REGION Network 73: Reset CMS
   // Reset Axis when the unit is in the resetting state.
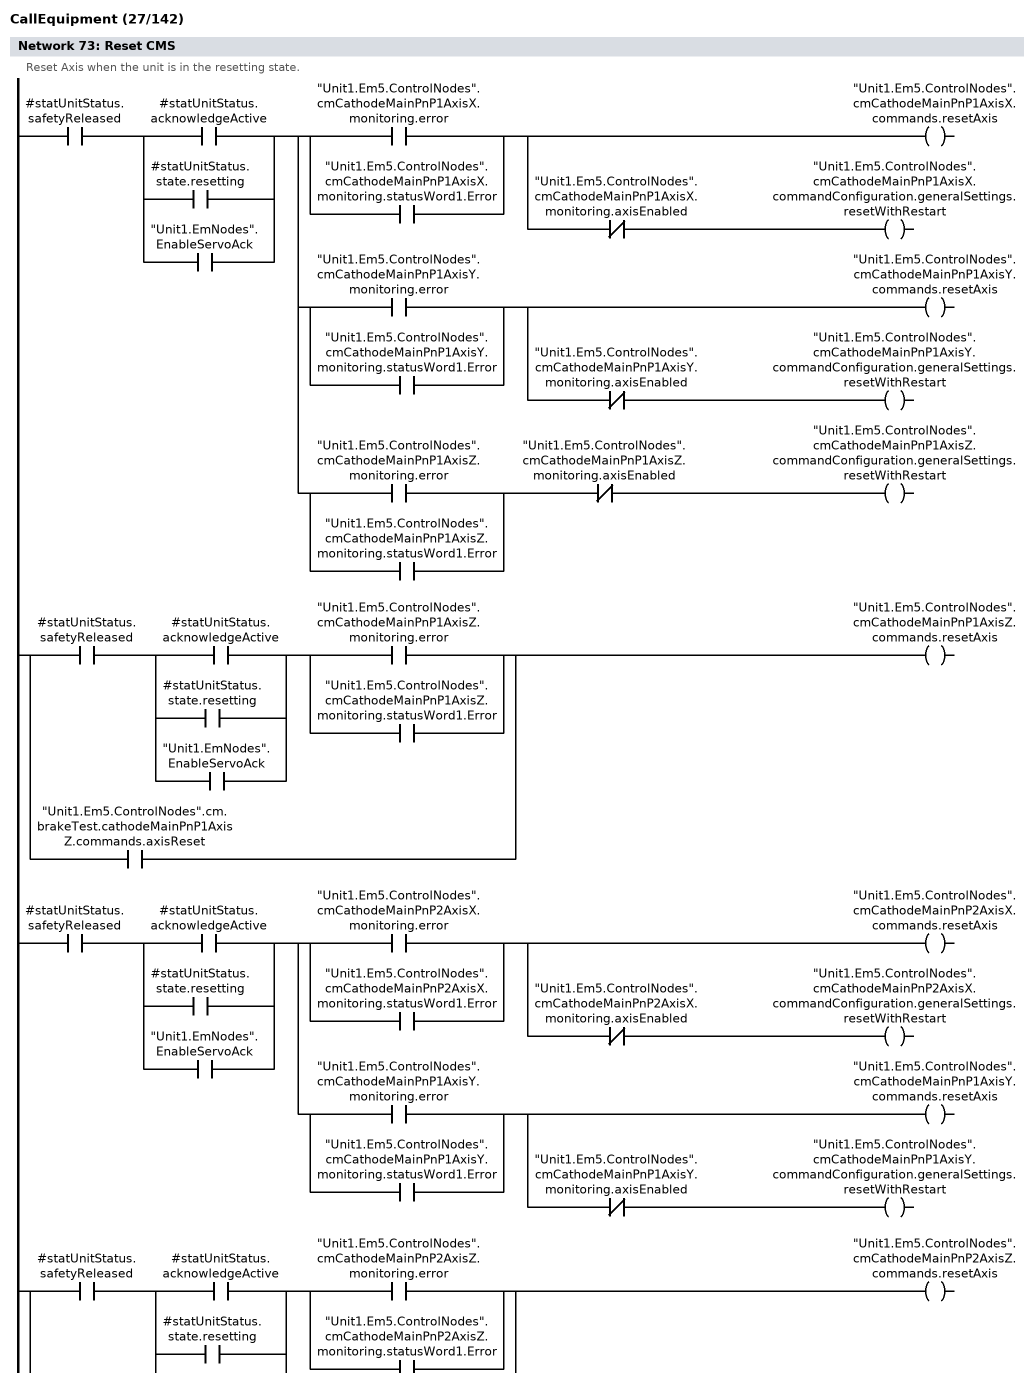
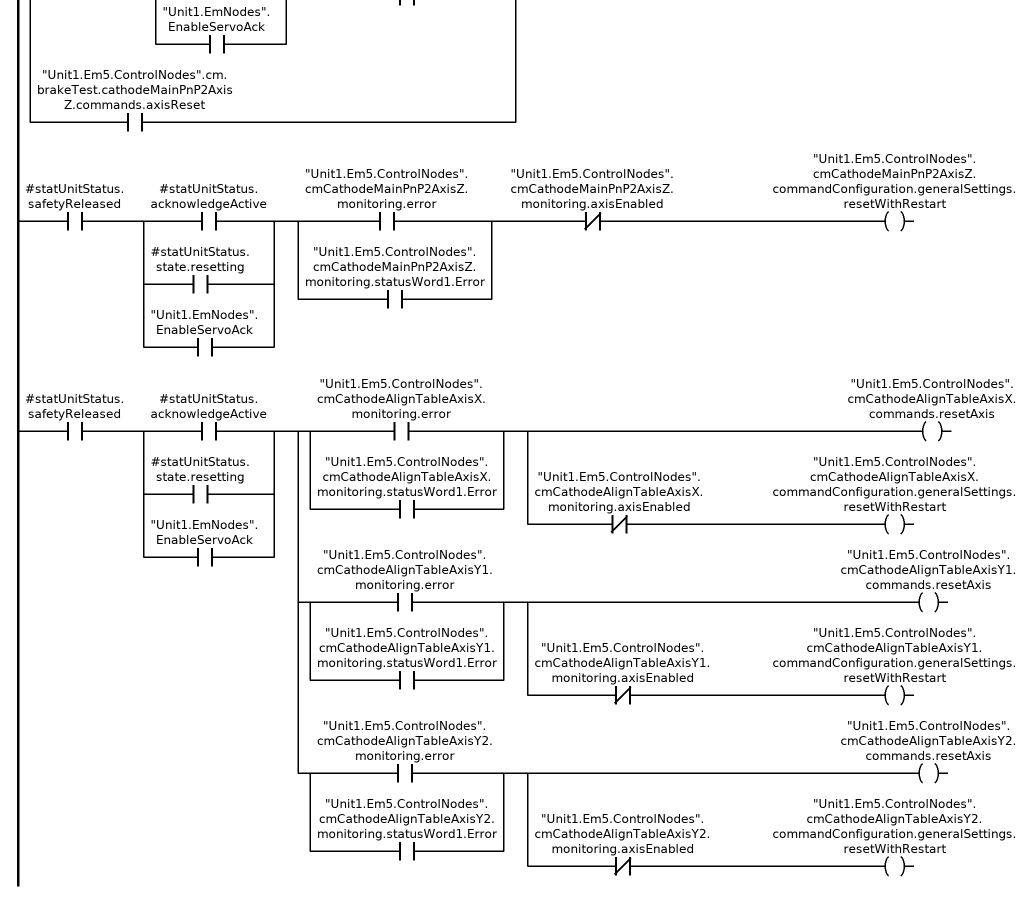
   RUNG wire#powerrail
      Contact( #statUnitStatus.safetyReleased )
      wire#w1
      Contact( #statUnitStatus.acknowledgeActive )
      wire#w2
      Contact( "Unit1.Em5.ControlNodes".cmCathodeMainPnP1AxisX.monitoring.error )
      wire#w3
      Coil( "Unit1.Em5.ControlNodes".cmCathodeMainPnP1AxisX.commands.resetAxis )
   END_RUNG
   RUNG wire#w1
      Contact( #statUnitStatus.state.resetting )
   END_RUNG wire#w2
   RUNG wire#w1
      Contact( "Unit1.EmNodes".EnableServoAck )
   END_RUNG wire#w2
   RUNG wire#w2
      Contact( "Unit1.Em5.ControlNodes".cmCathodeMainPnP1AxisX.monitoring.statusWord1.Error )
   END_RUNG wire#w3
   RUNG wire#w3
      I_Contact( "Unit1.Em5.ControlNodes".cmCathodeMainPnP1AxisX.monitoring.axisEnabled )
      Coil( "Unit1.Em5.ControlNodes".cmCathodeMainPnP1AxisX.commandConfiguration.generalSettings.resetWithRestart )
   END_RUNG
   RUNG wire#w2
      Contact( "Unit1.Em5.ControlNodes".cmCathodeMainPnP1AxisY.monitoring.error )
      wire#w4
      Coil( "Unit1.Em5.ControlNodes".cmCathodeMainPnP1AxisY.commands.resetAxis )
   END_RUNG
   RUNG wire#w2
      Contact( "Unit1.Em5.ControlNodes".cmCathodeMainPnP1AxisY.monitoring.statusWord1.Error )
   END_RUNG wire#w4
   RUNG wire#w4
      I_Contact( "Unit1.Em5.ControlNodes".cmCathodeMainPnP1AxisY.monitoring.axisEnabled )
      Coil( "Unit1.Em5.ControlNodes".cmCathodeMainPnP1AxisY.commandConfiguration.generalSettings.resetWithRestart )
   END_RUNG
   RUNG wire#w2
      Contact( "Unit1.Em5.ControlNodes".cmCathodeMainPnP1AxisZ.monitoring.error )
      wire#w5
      I_Contact( "Unit1.Em5.ControlNodes".cmCathodeMainPnP1AxisZ.monitoring.axisEnabled )
      Coil( "Unit1.Em5.ControlNodes".cmCathodeMainPnP1AxisZ.commandConfiguration.generalSettings.resetWithRestart )
   END_RUNG
   RUNG wire#w2
      Contact( "Unit1.Em5.ControlNodes".cmCathodeMainPnP1AxisZ.monitoring.statusWord1.Error )
   END_RUNG wire#w5
   RUNG wire#powerrail
      Contact( #statUnitStatus.safetyReleased )
      wire#w6
      Contact( #statUnitStatus.acknowledgeActive )
      wire#w7
      Contact( "Unit1.Em5.ControlNodes".cmCathodeMainPnP1AxisZ.monitoring.error )
      wire#w8
      Coil( "Unit1.Em5.ControlNodes".cmCathodeMainPnP1AxisZ.commands.resetAxis )
   END_RUNG
   RUNG wire#w6
      Contact( #statUnitStatus.state.resetting )
   END_RUNG wire#w7
   RUNG wire#w6
      Contact( "Unit1.EmNodes".EnableServoAck )
   END_RUNG wire#w7
   RUNG wire#w7
      Contact( "Unit1.Em5.ControlNodes".cmCathodeMainPnP1AxisZ.monitoring.statusWord1.Error )
   END_RUNG wire#w8
   RUNG wire#powerrail
      Contact( "Unit1.Em5.ControlNodes".cm.brakeTest.cathodeMainPnP1AxisZ.commands.axisReset )
   END_RUNG wire#w8
   RUNG wire#powerrail
      Contact( #statUnitStatus.safetyReleased )
      wire#w9
      Contact( #statUnitStatus.acknowledgeActive )
      wire#w10
      Contact( "Unit1.Em5.ControlNodes".cmCathodeMainPnP2AxisX.monitoring.error )
      wire#w11
      Coil( "Unit1.Em5.ControlNodes".cmCathodeMainPnP2AxisX.commands.resetAxis )
   END_RUNG
   RUNG wire#w9
      Contact( #statUnitStatus.state.resetting )
   END_RUNG wire#w10
   RUNG wire#w9
      Contact( "Unit1.EmNodes".EnableServoAck )
   END_RUNG wire#w10
   RUNG wire#w10
      Contact( "Unit1.Em5.ControlNodes".cmCathodeMainPnP2AxisX.monitoring.statusWord1.Error )
   END_RUNG wire#w11
   RUNG wire#w11
      I_Contact( "Unit1.Em5.ControlNodes".cmCathodeMainPnP2AxisX.monitoring.axisEnabled )
      Coil( "Unit1.Em5.ControlNodes".cmCathodeMainPnP2AxisX.commandConfiguration.generalSettings.resetWithRestart )
   END_RUNG
   RUNG wire#w10
      Contact( "Unit1.Em5.ControlNodes".cmCathodeMainPnP1AxisY.monitoring.error )
      wire#w12
      Coil( "Unit1.Em5.ControlNodes".cmCathodeMainPnP1AxisY.commands.resetAxis )
   END_RUNG
   RUNG wire#w10
      Contact( "Unit1.Em5.ControlNodes".cmCathodeMainPnP1AxisY.monitoring.statusWord1.Error )
   END_RUNG wire#w12
   RUNG wire#w12
      I_Contact( "Unit1.Em5.ControlNodes".cmCathodeMainPnP1AxisY.monitoring.axisEnabled )
      Coil( "Unit1.Em5.ControlNodes".cmCathodeMainPnP1AxisY.commandConfiguration.generalSettings.resetWithRestart )
   END_RUNG
   RUNG wire#powerrail
      Contact( #statUnitStatus.safetyReleased )
      wire#w13
      Contact( #statUnitStatus.acknowledgeActive )
      wire#w14
      Contact( "Unit1.Em5.ControlNodes".cmCathodeMainPnP2AxisZ.monitoring.error )
      wire#w15
      Coil( "Unit1.Em5.ControlNodes".cmCathodeMainPnP2AxisZ.commands.resetAxis )
   END_RUNG
   RUNG wire#w13
      Contact( #statUnitStatus.state.resetting )
   END_RUNG wire#w14
   RUNG wire#w13
      Contact( "Unit1.EmNodes".EnableServoAck )
   END_RUNG wire#w14
   RUNG wire#w14
      Contact( "Unit1.Em5.ControlNodes".cmCathodeMainPnP2AxisZ.monitoring.statusWord1.Error )
   END_RUNG wire#w15
   RUNG wire#powerrail
      Contact( "Unit1.Em5.ControlNodes".cm.brakeTest.cathodeMainPnP2AxisZ.commands.axisReset )
   END_RUNG wire#w15
   RUNG wire#powerrail
      Contact( #statUnitStatus.safetyReleased )
      wire#w16
      Contact( #statUnitStatus.acknowledgeActive )
      wire#w17
      Contact( "Unit1.Em5.ControlNodes".cmCathodeMainPnP2AxisZ.monitoring.error )
      wire#w18
      I_Contact( "Unit1.Em5.ControlNodes".cmCathodeMainPnP2AxisZ.monitoring.axisEnabled )
      Coil( "Unit1.Em5.ControlNodes".cmCathodeMainPnP2AxisZ.commandConfiguration.generalSettings.resetWithRestart )
   END_RUNG
   RUNG wire#w16
      Contact( #statUnitStatus.state.resetting )
   END_RUNG wire#w17
   RUNG wire#w16
      Contact( "Unit1.EmNodes".EnableServoAck )
   END_RUNG wire#w17
   RUNG wire#w17
      Contact( "Unit1.Em5.ControlNodes".cmCathodeMainPnP2AxisZ.monitoring.statusWord1.Error )
   END_RUNG wire#w18
   RUNG wire#powerrail
      Contact( #statUnitStatus.safetyReleased )
      wire#w19
      Contact( #statUnitStatus.acknowledgeActive )
      wire#w20
      Contact( "Unit1.Em5.ControlNodes".cmCathodeAlignTableAxisX.monitoring.error )
      wire#w21
      Coil( "Unit1.Em5.ControlNodes".cmCathodeAlignTableAxisX.commands.resetAxis )
   END_RUNG
   RUNG wire#w19
      Contact( #statUnitStatus.state.resetting )
   END_RUNG wire#w20
   RUNG wire#w19
      Contact( "Unit1.EmNodes".EnableServoAck )
   END_RUNG wire#w20
   RUNG wire#w20
      Contact( "Unit1.Em5.ControlNodes".cmCathodeAlignTableAxisX.monitoring.statusWord1.Error )
   END_RUNG wire#w21
   RUNG wire#w21
      I_Contact( "Unit1.Em5.ControlNodes".cmCathodeAlignTableAxisX.monitoring.axisEnabled )
      Coil( "Unit1.Em5.ControlNodes".cmCathodeAlignTableAxisX.commandConfiguration.generalSettings.resetWithRestart )
   END_RUNG
   RUNG wire#w20
      Contact( "Unit1.Em5.ControlNodes".cmCathodeAlignTableAxisY1.monitoring.error )
      wire#w22
      Coil( "Unit1.Em5.ControlNodes".cmCathodeAlignTableAxisY1.commands.resetAxis )
   END_RUNG
   RUNG wire#w20
      Contact( "Unit1.Em5.ControlNodes".cmCathodeAlignTableAxisY1.monitoring.statusWord1.Error )
   END_RUNG wire#w22
   RUNG wire#w22
      I_Contact( "Unit1.Em5.ControlNodes".cmCathodeAlignTableAxisY1.monitoring.axisEnabled )
      Coil( "Unit1.Em5.ControlNodes".cmCathodeAlignTableAxisY1.commandConfiguration.generalSettings.resetWithRestart )
   END_RUNG
   RUNG wire#w20
      Contact( "Unit1.Em5.ControlNodes".cmCathodeAlignTableAxisY2.monitoring.error )
      wire#w23
      Coil( "Unit1.Em5.ControlNodes".cmCathodeAlignTableAxisY2.commands.resetAxis )
   END_RUNG
   RUNG wire#w20
      Contact( "Unit1.Em5.ControlNodes".cmCathodeAlignTableAxisY2.monitoring.statusWord1.Error )
   END_RUNG wire#w23
   RUNG wire#w23
      I_Contact( "Unit1.Em5.ControlNodes".cmCathodeAlignTableAxisY2.monitoring.axisEnabled )
      Coil( "Unit1.Em5.ControlNodes".cmCathodeAlignTableAxisY2.commandConfiguration.generalSettings.resetWithRestart )
   END_RUNG
   // the same network as SCL:
   #_w1 := #statUnitStatus.safetyReleased AND (#statUnitStatus.acknowledgeActive OR #statUnitStatus.state.resetting OR "Unit1.EmNodes".EnableServoAck);
   "Unit1.Em5.ControlNodes".cmCathodeMainPnP1AxisX.commands.resetAxis := #_w1 AND ("Unit1.Em5.ControlNodes".cmCathodeMainPnP1AxisX.monitoring.error OR "Unit1.Em5.ControlNodes".cmCathodeMainPnP1AxisX.monitoring.statusWord1.Error);
   "Unit1.Em5.ControlNodes".cmCathodeMainPnP1AxisX.commandConfiguration.generalSettings.resetWithRestart := "Unit1.Em5.ControlNodes".cmCathodeMainPnP1AxisX.commands.resetAxis AND NOT "Unit1.Em5.ControlNodes".cmCathodeMainPnP1AxisX.monitoring.axisEnabled;
   "Unit1.Em5.ControlNodes".cmCathodeMainPnP1AxisY.commands.resetAxis := #_w1 AND ("Unit1.Em5.ControlNodes".cmCathodeMainPnP1AxisY.monitoring.error OR "Unit1.Em5.ControlNodes".cmCathodeMainPnP1AxisY.monitoring.statusWord1.Error);
   "Unit1.Em5.ControlNodes".cmCathodeMainPnP1AxisY.commandConfiguration.generalSettings.resetWithRestart := "Unit1.Em5.ControlNodes".cmCathodeMainPnP1AxisY.commands.resetAxis AND NOT "Unit1.Em5.ControlNodes".cmCathodeMainPnP1AxisY.monitoring.axisEnabled;
   "Unit1.Em5.ControlNodes".cmCathodeMainPnP1AxisZ.commandConfiguration.generalSettings.resetWithRestart := #_w1 AND ("Unit1.Em5.ControlNodes".cmCathodeMainPnP1AxisZ.monitoring.error OR "Unit1.Em5.ControlNodes".cmCathodeMainPnP1AxisZ.monitoring.statusWord1.Error) AND NOT "Unit1.Em5.ControlNodes".cmCathodeMainPnP1AxisZ.monitoring.axisEnabled;
   "Unit1.Em5.ControlNodes".cmCathodeMainPnP1AxisZ.commands.resetAxis := (#statUnitStatus.safetyReleased AND (#statUnitStatus.acknowledgeActive OR #statUnitStatus.state.resetting OR "Unit1.EmNodes".EnableServoAck) AND ("Unit1.Em5.ControlNodes".cmCathodeMainPnP1AxisZ.monitoring.error OR "Unit1.Em5.ControlNodes".cmCathodeMainPnP1AxisZ.monitoring.statusWord1.Error)) OR "Unit1.Em5.ControlNodes".cm.brakeTest.cathodeMainPnP1AxisZ.commands.axisReset;
   #_w2 := #statUnitStatus.safetyReleased AND (#statUnitStatus.acknowledgeActive OR #statUnitStatus.state.resetting OR "Unit1.EmNodes".EnableServoAck);
   "Unit1.Em5.ControlNodes".cmCathodeMainPnP2AxisX.commands.resetAxis := #_w2 AND ("Unit1.Em5.ControlNodes".cmCathodeMainPnP2AxisX.monitoring.error OR "Unit1.Em5.ControlNodes".cmCathodeMainPnP2AxisX.monitoring.statusWord1.Error);
   "Unit1.Em5.ControlNodes".cmCathodeMainPnP2AxisX.commandConfiguration.generalSettings.resetWithRestart := "Unit1.Em5.ControlNodes".cmCathodeMainPnP2AxisX.commands.resetAxis AND NOT "Unit1.Em5.ControlNodes".cmCathodeMainPnP2AxisX.monitoring.axisEnabled;
   "Unit1.Em5.ControlNodes".cmCathodeMainPnP1AxisY.commands.resetAxis := #_w2 AND ("Unit1.Em5.ControlNodes".cmCathodeMainPnP1AxisY.monitoring.error OR "Unit1.Em5.ControlNodes".cmCathodeMainPnP1AxisY.monitoring.statusWord1.Error);
   "Unit1.Em5.ControlNodes".cmCathodeMainPnP1AxisY.commandConfiguration.generalSettings.resetWithRestart := "Unit1.Em5.ControlNodes".cmCathodeMainPnP1AxisY.commands.resetAxis AND NOT "Unit1.Em5.ControlNodes".cmCathodeMainPnP1AxisY.monitoring.axisEnabled;
   "Unit1.Em5.ControlNodes".cmCathodeMainPnP2AxisZ.commands.resetAxis := (#statUnitStatus.safetyReleased AND (#statUnitStatus.acknowledgeActive OR #statUnitStatus.state.resetting OR "Unit1.EmNodes".EnableServoAck) AND ("Unit1.Em5.ControlNodes".cmCathodeMainPnP2AxisZ.monitoring.error OR "Unit1.Em5.ControlNodes".cmCathodeMainPnP2AxisZ.monitoring.statusWord1.Error)) OR "Unit1.Em5.ControlNodes".cm.brakeTest.cathodeMainPnP2AxisZ.commands.axisReset;
   "Unit1.Em5.ControlNodes".cmCathodeMainPnP2AxisZ.commandConfiguration.generalSettings.resetWithRestart := #statUnitStatus.safetyReleased AND (#statUnitStatus.acknowledgeActive OR #statUnitStatus.state.resetting OR "Unit1.EmNodes".EnableServoAck) AND ("Unit1.Em5.ControlNodes".cmCathodeMainPnP2AxisZ.monitoring.error OR "Unit1.Em5.ControlNodes".cmCathodeMainPnP2AxisZ.monitoring.statusWord1.Error) AND NOT "Unit1.Em5.ControlNodes".cmCathodeMainPnP2AxisZ.monitoring.axisEnabled;
   #_w3 := #statUnitStatus.safetyReleased AND (#statUnitStatus.acknowledgeActive OR #statUnitStatus.state.resetting OR "Unit1.EmNodes".EnableServoAck);
   "Unit1.Em5.ControlNodes".cmCathodeAlignTableAxisX.commands.resetAxis := #_w3 AND ("Unit1.Em5.ControlNodes".cmCathodeAlignTableAxisX.monitoring.error OR "Unit1.Em5.ControlNodes".cmCathodeAlignTableAxisX.monitoring.statusWord1.Error);
   "Unit1.Em5.ControlNodes".cmCathodeAlignTableAxisX.commandConfiguration.generalSettings.resetWithRestart := "Unit1.Em5.ControlNodes".cmCathodeAlignTableAxisX.commands.resetAxis AND NOT "Unit1.Em5.ControlNodes".cmCathodeAlignTableAxisX.monitoring.axisEnabled;
   "Unit1.Em5.ControlNodes".cmCathodeAlignTableAxisY1.commands.resetAxis := #_w3 AND ("Unit1.Em5.ControlNodes".cmCathodeAlignTableAxisY1.monitoring.error OR "Unit1.Em5.ControlNodes".cmCathodeAlignTableAxisY1.monitoring.statusWord1.Error);
   "Unit1.Em5.ControlNodes".cmCathodeAlignTableAxisY1.commandConfiguration.generalSettings.resetWithRestart := "Unit1.Em5.ControlNodes".cmCathodeAlignTableAxisY1.commands.resetAxis AND NOT "Unit1.Em5.ControlNodes".cmCathodeAlignTableAxisY1.monitoring.axisEnabled;
   "Unit1.Em5.ControlNodes".cmCathodeAlignTableAxisY2.commands.resetAxis := #_w3 AND ("Unit1.Em5.ControlNodes".cmCathodeAlignTableAxisY2.monitoring.error OR "Unit1.Em5.ControlNodes".cmCathodeAlignTableAxisY2.monitoring.statusWord1.Error);
   "Unit1.Em5.ControlNodes".cmCathodeAlignTableAxisY2.commandConfiguration.generalSettings.resetWithRestart := "Unit1.Em5.ControlNodes".cmCathodeAlignTableAxisY2.commands.resetAxis AND NOT "Unit1.Em5.ControlNodes".cmCathodeAlignTableAxisY2.monitoring.axisEnabled;
END_REGION

REGION Network 74: Enable/Disable CMs
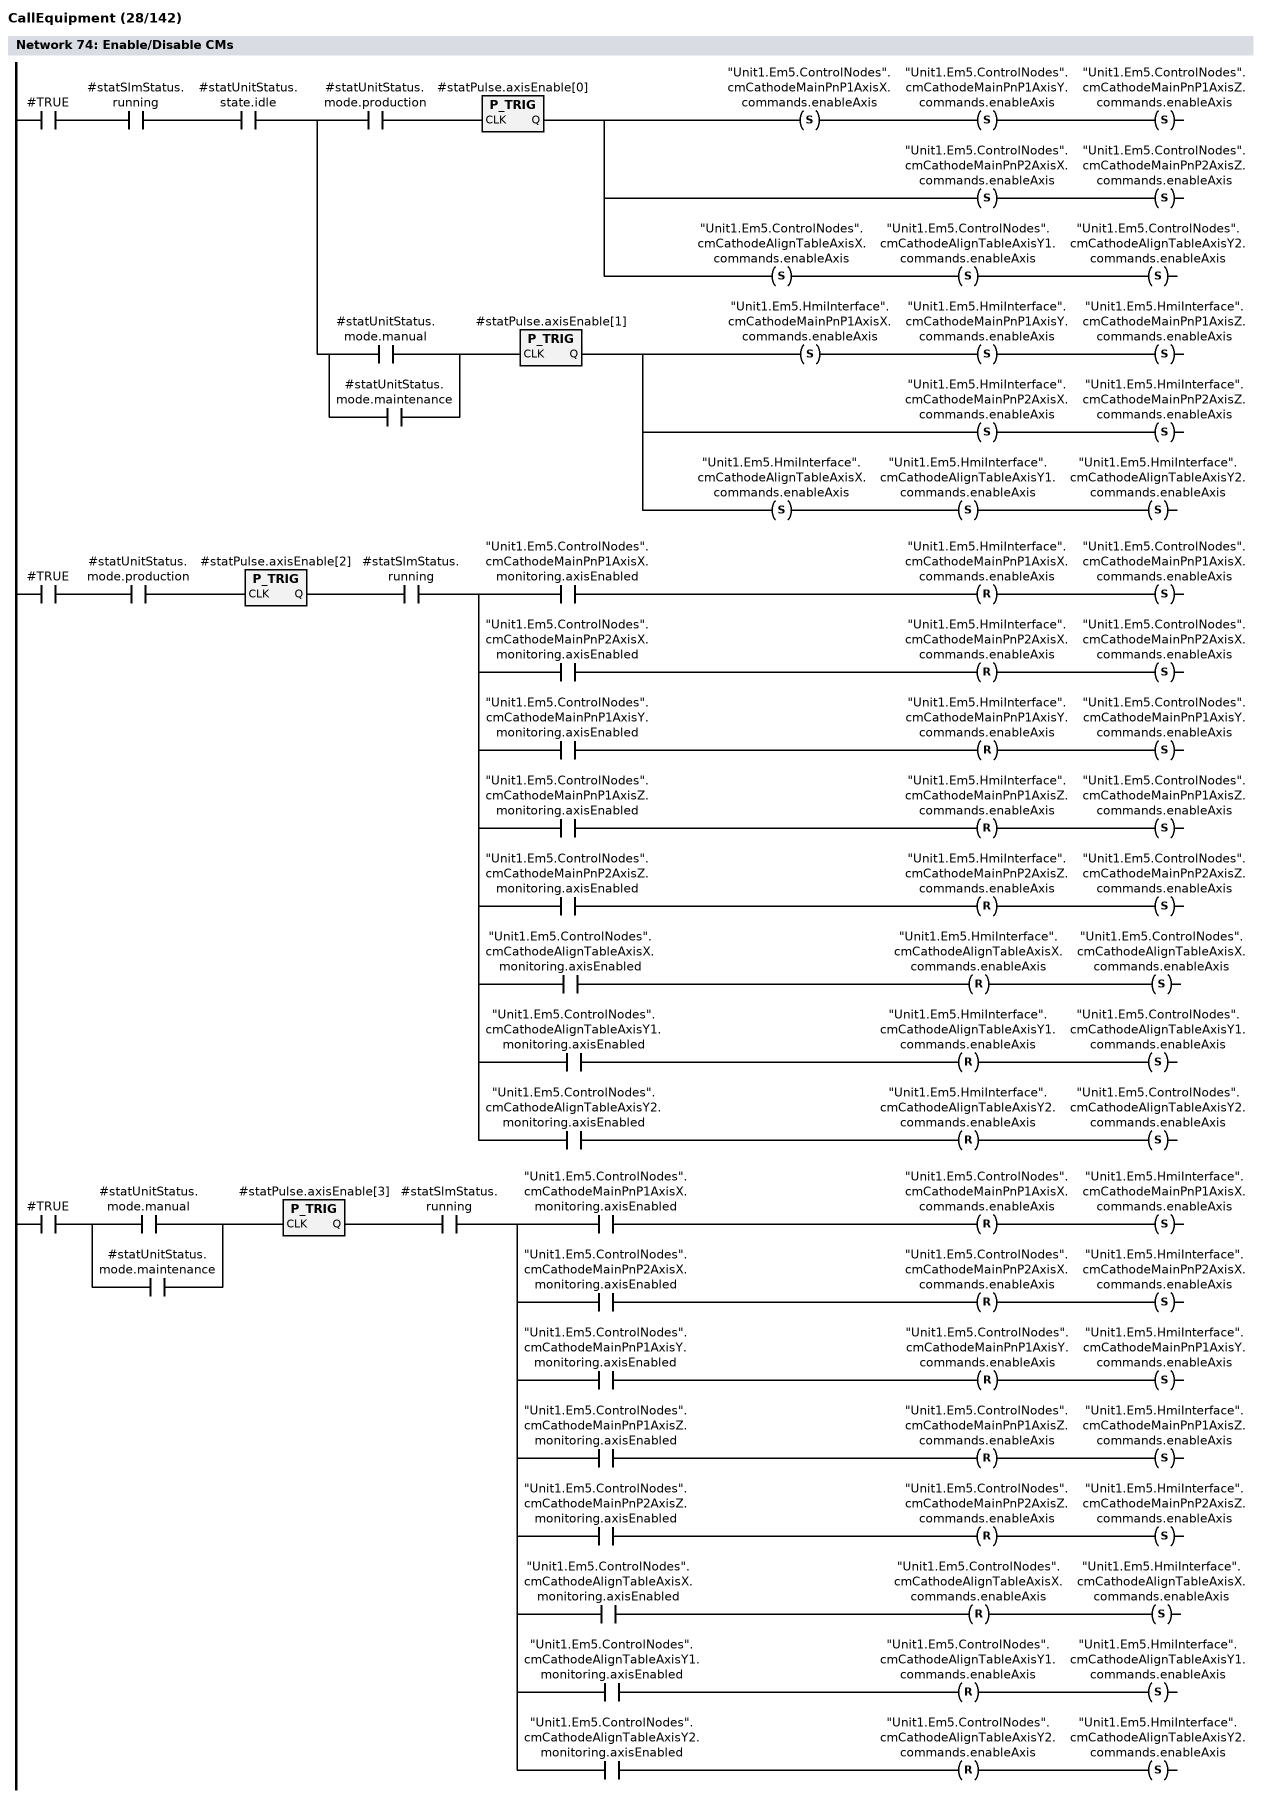
   RUNG wire#powerrail
      Contact( #TRUE )
      Contact( #statSlmStatus.running )
      Contact( #statUnitStatus.state.idle )
      wire#w1
      Contact( #statUnitStatus.mode.production )
      P_Trig( #statPulse.axisEnable[0] )
      wire#w2
      S_Coil( "Unit1.Em5.ControlNodes".cmCathodeMainPnP1AxisX.commands.enableAxis )
      S_Coil( "Unit1.Em5.ControlNodes".cmCathodeMainPnP1AxisY.commands.enableAxis )
      S_Coil( "Unit1.Em5.ControlNodes".cmCathodeMainPnP1AxisZ.commands.enableAxis )
   END_RUNG
   RUNG wire#w2
      S_Coil( "Unit1.Em5.ControlNodes".cmCathodeMainPnP2AxisX.commands.enableAxis )
      S_Coil( "Unit1.Em5.ControlNodes".cmCathodeMainPnP2AxisZ.commands.enableAxis )
   END_RUNG
   RUNG wire#w2
      S_Coil( "Unit1.Em5.ControlNodes".cmCathodeAlignTableAxisX.commands.enableAxis )
      S_Coil( "Unit1.Em5.ControlNodes".cmCathodeAlignTableAxisY1.commands.enableAxis )
      S_Coil( "Unit1.Em5.ControlNodes".cmCathodeAlignTableAxisY2.commands.enableAxis )
   END_RUNG
   RUNG wire#w1
      Contact( #statUnitStatus.mode.manual )
      wire#w3
      P_Trig( #statPulse.axisEnable[1] )
      wire#w4
      S_Coil( "Unit1.Em5.HmiInterface".cmCathodeMainPnP1AxisX.commands.enableAxis )
      S_Coil( "Unit1.Em5.HmiInterface".cmCathodeMainPnP1AxisY.commands.enableAxis )
      S_Coil( "Unit1.Em5.HmiInterface".cmCathodeMainPnP1AxisZ.commands.enableAxis )
   END_RUNG
   RUNG wire#w1
      Contact( #statUnitStatus.mode.maintenance )
   END_RUNG wire#w3
   RUNG wire#w4
      S_Coil( "Unit1.Em5.HmiInterface".cmCathodeMainPnP2AxisX.commands.enableAxis )
      S_Coil( "Unit1.Em5.HmiInterface".cmCathodeMainPnP2AxisZ.commands.enableAxis )
   END_RUNG
   RUNG wire#w4
      S_Coil( "Unit1.Em5.HmiInterface".cmCathodeAlignTableAxisX.commands.enableAxis )
      S_Coil( "Unit1.Em5.HmiInterface".cmCathodeAlignTableAxisY1.commands.enableAxis )
      S_Coil( "Unit1.Em5.HmiInterface".cmCathodeAlignTableAxisY2.commands.enableAxis )
   END_RUNG
   RUNG wire#powerrail
      Contact( #TRUE )
      Contact( #statUnitStatus.mode.production )
      P_Trig( #statPulse.axisEnable[2] )
      Contact( #statSlmStatus.running )
      wire#w5
      Contact( "Unit1.Em5.ControlNodes".cmCathodeMainPnP1AxisX.monitoring.axisEnabled )
      R_Coil( "Unit1.Em5.HmiInterface".cmCathodeMainPnP1AxisX.commands.enableAxis )
      S_Coil( "Unit1.Em5.ControlNodes".cmCathodeMainPnP1AxisX.commands.enableAxis )
   END_RUNG
   RUNG wire#w5
      Contact( "Unit1.Em5.ControlNodes".cmCathodeMainPnP2AxisX.monitoring.axisEnabled )
      R_Coil( "Unit1.Em5.HmiInterface".cmCathodeMainPnP2AxisX.commands.enableAxis )
      S_Coil( "Unit1.Em5.ControlNodes".cmCathodeMainPnP2AxisX.commands.enableAxis )
   END_RUNG
   RUNG wire#w5
      Contact( "Unit1.Em5.ControlNodes".cmCathodeMainPnP1AxisY.monitoring.axisEnabled )
      R_Coil( "Unit1.Em5.HmiInterface".cmCathodeMainPnP1AxisY.commands.enableAxis )
      S_Coil( "Unit1.Em5.ControlNodes".cmCathodeMainPnP1AxisY.commands.enableAxis )
   END_RUNG
   RUNG wire#w5
      Contact( "Unit1.Em5.ControlNodes".cmCathodeMainPnP1AxisZ.monitoring.axisEnabled )
      R_Coil( "Unit1.Em5.HmiInterface".cmCathodeMainPnP1AxisZ.commands.enableAxis )
      S_Coil( "Unit1.Em5.ControlNodes".cmCathodeMainPnP1AxisZ.commands.enableAxis )
   END_RUNG
   RUNG wire#w5
      Contact( "Unit1.Em5.ControlNodes".cmCathodeMainPnP2AxisZ.monitoring.axisEnabled )
      R_Coil( "Unit1.Em5.HmiInterface".cmCathodeMainPnP2AxisZ.commands.enableAxis )
      S_Coil( "Unit1.Em5.ControlNodes".cmCathodeMainPnP2AxisZ.commands.enableAxis )
   END_RUNG
   RUNG wire#w5
      Contact( "Unit1.Em5.ControlNodes".cmCathodeAlignTableAxisX.monitoring.axisEnabled )
      R_Coil( "Unit1.Em5.HmiInterface".cmCathodeAlignTableAxisX.commands.enableAxis )
      S_Coil( "Unit1.Em5.ControlNodes".cmCathodeAlignTableAxisX.commands.enableAxis )
   END_RUNG
   RUNG wire#w5
      Contact( "Unit1.Em5.ControlNodes".cmCathodeAlignTableAxisY1.monitoring.axisEnabled )
      R_Coil( "Unit1.Em5.HmiInterface".cmCathodeAlignTableAxisY1.commands.enableAxis )
      S_Coil( "Unit1.Em5.ControlNodes".cmCathodeAlignTableAxisY1.commands.enableAxis )
   END_RUNG
   RUNG wire#w5
      Contact( "Unit1.Em5.ControlNodes".cmCathodeAlignTableAxisY2.monitoring.axisEnabled )
      R_Coil( "Unit1.Em5.HmiInterface".cmCathodeAlignTableAxisY2.commands.enableAxis )
      S_Coil( "Unit1.Em5.ControlNodes".cmCathodeAlignTableAxisY2.commands.enableAxis )
   END_RUNG
   RUNG wire#powerrail
      Contact( #TRUE )
      wire#w6
      Contact( #statUnitStatus.mode.manual )
      wire#w7
      P_Trig( #statPulse.axisEnable[3] )
      Contact( #statSlmStatus.running )
      wire#w8
      Contact( "Unit1.Em5.ControlNodes".cmCathodeMainPnP1AxisX.monitoring.axisEnabled )
      R_Coil( "Unit1.Em5.ControlNodes".cmCathodeMainPnP1AxisX.commands.enableAxis )
      S_Coil( "Unit1.Em5.HmiInterface".cmCathodeMainPnP1AxisX.commands.enableAxis )
   END_RUNG
   RUNG wire#w6
      Contact( #statUnitStatus.mode.maintenance )
   END_RUNG wire#w7
   RUNG wire#w8
      Contact( "Unit1.Em5.ControlNodes".cmCathodeMainPnP2AxisX.monitoring.axisEnabled )
      R_Coil( "Unit1.Em5.ControlNodes".cmCathodeMainPnP2AxisX.commands.enableAxis )
      S_Coil( "Unit1.Em5.HmiInterface".cmCathodeMainPnP2AxisX.commands.enableAxis )
   END_RUNG
   RUNG wire#w8
      Contact( "Unit1.Em5.ControlNodes".cmCathodeMainPnP1AxisY.monitoring.axisEnabled )
      R_Coil( "Unit1.Em5.ControlNodes".cmCathodeMainPnP1AxisY.commands.enableAxis )
      S_Coil( "Unit1.Em5.HmiInterface".cmCathodeMainPnP1AxisY.commands.enableAxis )
   END_RUNG
   RUNG wire#w8
      Contact( "Unit1.Em5.ControlNodes".cmCathodeMainPnP1AxisZ.monitoring.axisEnabled )
      R_Coil( "Unit1.Em5.ControlNodes".cmCathodeMainPnP1AxisZ.commands.enableAxis )
      S_Coil( "Unit1.Em5.HmiInterface".cmCathodeMainPnP1AxisZ.commands.enableAxis )
   END_RUNG
   RUNG wire#w8
      Contact( "Unit1.Em5.ControlNodes".cmCathodeMainPnP2AxisZ.monitoring.axisEnabled )
      R_Coil( "Unit1.Em5.ControlNodes".cmCathodeMainPnP2AxisZ.commands.enableAxis )
      S_Coil( "Unit1.Em5.HmiInterface".cmCathodeMainPnP2AxisZ.commands.enableAxis )
   END_RUNG
   RUNG wire#w8
      Contact( "Unit1.Em5.ControlNodes".cmCathodeAlignTableAxisX.monitoring.axisEnabled )
      R_Coil( "Unit1.Em5.ControlNodes".cmCathodeAlignTableAxisX.commands.enableAxis )
      S_Coil( "Unit1.Em5.HmiInterface".cmCathodeAlignTableAxisX.commands.enableAxis )
   END_RUNG
   RUNG wire#w8
      Contact( "Unit1.Em5.ControlNodes".cmCathodeAlignTableAxisY1.monitoring.axisEnabled )
      R_Coil( "Unit1.Em5.ControlNodes".cmCathodeAlignTableAxisY1.commands.enableAxis )
      S_Coil( "Unit1.Em5.HmiInterface".cmCathodeAlignTableAxisY1.commands.enableAxis )
   END_RUNG
   RUNG wire#w8
      Contact( "Unit1.Em5.ControlNodes".cmCathodeAlignTableAxisY2.monitoring.axisEnabled )
      R_Coil( "Unit1.Em5.ControlNodes".cmCathodeAlignTableAxisY2.commands.enableAxis )
      S_Coil( "Unit1.Em5.HmiInterface".cmCathodeAlignTableAxisY2.commands.enableAxis )
   END_RUNG
   // the same network as SCL:
   #_w1 := #TRUE AND #statSlmStatus.running AND #statUnitStatus.state.idle;
   #_w2 := #_w1 AND #statUnitStatus.mode.production;
   #_w3 := #_w2 AND NOT #statPulse.axisEnable[0];   // rising edge
   #statPulse.axisEnable[0] := #_w2;
   IF #_w3 THEN
       "Unit1.Em5.ControlNodes".cmCathodeMainPnP1AxisX.commands.enableAxis := TRUE;
       "Unit1.Em5.ControlNodes".cmCathodeMainPnP1AxisY.commands.enableAxis := TRUE;
       "Unit1.Em5.ControlNodes".cmCathodeMainPnP1AxisZ.commands.enableAxis := TRUE;
       "Unit1.Em5.ControlNodes".cmCathodeMainPnP2AxisX.commands.enableAxis := TRUE;
       "Unit1.Em5.ControlNodes".cmCathodeMainPnP2AxisZ.commands.enableAxis := TRUE;
       "Unit1.Em5.ControlNodes".cmCathodeAlignTableAxisX.commands.enableAxis := TRUE;
       "Unit1.Em5.ControlNodes".cmCathodeAlignTableAxisY1.commands.enableAxis := TRUE;
       "Unit1.Em5.ControlNodes".cmCathodeAlignTableAxisY2.commands.enableAxis := TRUE;
   END_IF;
   #_w4 := #_w1 AND (#statUnitStatus.mode.manual OR #statUnitStatus.mode.maintenance);
   #_w5 := #_w4 AND NOT #statPulse.axisEnable[1];   // rising edge
   #statPulse.axisEnable[1] := #_w4;
   IF #_w5 THEN
       "Unit1.Em5.HmiInterface".cmCathodeMainPnP1AxisX.commands.enableAxis := TRUE;
       "Unit1.Em5.HmiInterface".cmCathodeMainPnP1AxisY.commands.enableAxis := TRUE;
       "Unit1.Em5.HmiInterface".cmCathodeMainPnP1AxisZ.commands.enableAxis := TRUE;
       "Unit1.Em5.HmiInterface".cmCathodeMainPnP2AxisX.commands.enableAxis := TRUE;
       "Unit1.Em5.HmiInterface".cmCathodeMainPnP2AxisZ.commands.enableAxis := TRUE;
       "Unit1.Em5.HmiInterface".cmCathodeAlignTableAxisX.commands.enableAxis := TRUE;
       "Unit1.Em5.HmiInterface".cmCathodeAlignTableAxisY1.commands.enableAxis := TRUE;
       "Unit1.Em5.HmiInterface".cmCathodeAlignTableAxisY2.commands.enableAxis := TRUE;
   END_IF;
   #_w6 := #TRUE AND #statUnitStatus.mode.production;
   #_w7 := #_w6 AND NOT #statPulse.axisEnable[2];   // rising edge
   #statPulse.axisEnable[2] := #_w6;
   #_w8 := #_w7 AND #statSlmStatus.running;
   IF #_w8 AND "Unit1.Em5.ControlNodes".cmCathodeMainPnP1AxisX.monitoring.axisEnabled THEN
       "Unit1.Em5.HmiInterface".cmCathodeMainPnP1AxisX.commands.enableAxis := FALSE;
       "Unit1.Em5.ControlNodes".cmCathodeMainPnP1AxisX.commands.enableAxis := TRUE;
   END_IF;
   IF #_w8 AND "Unit1.Em5.ControlNodes".cmCathodeMainPnP2AxisX.monitoring.axisEnabled THEN
       "Unit1.Em5.HmiInterface".cmCathodeMainPnP2AxisX.commands.enableAxis := FALSE;
       "Unit1.Em5.ControlNodes".cmCathodeMainPnP2AxisX.commands.enableAxis := TRUE;
   END_IF;
   IF #_w8 AND "Unit1.Em5.ControlNodes".cmCathodeMainPnP1AxisY.monitoring.axisEnabled THEN
       "Unit1.Em5.HmiInterface".cmCathodeMainPnP1AxisY.commands.enableAxis := FALSE;
       "Unit1.Em5.ControlNodes".cmCathodeMainPnP1AxisY.commands.enableAxis := TRUE;
   END_IF;
   IF #_w8 AND "Unit1.Em5.ControlNodes".cmCathodeMainPnP1AxisZ.monitoring.axisEnabled THEN
       "Unit1.Em5.HmiInterface".cmCathodeMainPnP1AxisZ.commands.enableAxis := FALSE;
       "Unit1.Em5.ControlNodes".cmCathodeMainPnP1AxisZ.commands.enableAxis := TRUE;
   END_IF;
   IF #_w8 AND "Unit1.Em5.ControlNodes".cmCathodeMainPnP2AxisZ.monitoring.axisEnabled THEN
       "Unit1.Em5.HmiInterface".cmCathodeMainPnP2AxisZ.commands.enableAxis := FALSE;
       "Unit1.Em5.ControlNodes".cmCathodeMainPnP2AxisZ.commands.enableAxis := TRUE;
   END_IF;
   IF #_w8 AND "Unit1.Em5.ControlNodes".cmCathodeAlignTableAxisX.monitoring.axisEnabled THEN
       "Unit1.Em5.HmiInterface".cmCathodeAlignTableAxisX.commands.enableAxis := FALSE;
       "Unit1.Em5.ControlNodes".cmCathodeAlignTableAxisX.commands.enableAxis := TRUE;
   END_IF;
   IF #_w8 AND "Unit1.Em5.ControlNodes".cmCathodeAlignTableAxisY1.monitoring.axisEnabled THEN
       "Unit1.Em5.HmiInterface".cmCathodeAlignTableAxisY1.commands.enableAxis := FALSE;
       "Unit1.Em5.ControlNodes".cmCathodeAlignTableAxisY1.commands.enableAxis := TRUE;
   END_IF;
   IF #_w8 AND "Unit1.Em5.ControlNodes".cmCathodeAlignTableAxisY2.monitoring.axisEnabled THEN
       "Unit1.Em5.HmiInterface".cmCathodeAlignTableAxisY2.commands.enableAxis := FALSE;
       "Unit1.Em5.ControlNodes".cmCathodeAlignTableAxisY2.commands.enableAxis := TRUE;
   END_IF;
   #_w9 := #TRUE AND (#statUnitStatus.mode.manual OR #statUnitStatus.mode.maintenance);
   #_w10 := #_w9 AND NOT #statPulse.axisEnable[3];   // rising edge
   #statPulse.axisEnable[3] := #_w9;
   #_w11 := #_w10 AND #statSlmStatus.running;
   IF #_w11 AND "Unit1.Em5.ControlNodes".cmCathodeMainPnP1AxisX.monitoring.axisEnabled THEN
       "Unit1.Em5.ControlNodes".cmCathodeMainPnP1AxisX.commands.enableAxis := FALSE;
       "Unit1.Em5.HmiInterface".cmCathodeMainPnP1AxisX.commands.enableAxis := TRUE;
   END_IF;
   IF #_w11 AND "Unit1.Em5.ControlNodes".cmCathodeMainPnP2AxisX.monitoring.axisEnabled THEN
       "Unit1.Em5.ControlNodes".cmCathodeMainPnP2AxisX.commands.enableAxis := FALSE;
       "Unit1.Em5.HmiInterface".cmCathodeMainPnP2AxisX.commands.enableAxis := TRUE;
   END_IF;
   IF #_w11 AND "Unit1.Em5.ControlNodes".cmCathodeMainPnP1AxisY.monitoring.axisEnabled THEN
       "Unit1.Em5.ControlNodes".cmCathodeMainPnP1AxisY.commands.enableAxis := FALSE;
       "Unit1.Em5.HmiInterface".cmCathodeMainPnP1AxisY.commands.enableAxis := TRUE;
   END_IF;
   IF #_w11 AND "Unit1.Em5.ControlNodes".cmCathodeMainPnP1AxisZ.monitoring.axisEnabled THEN
       "Unit1.Em5.ControlNodes".cmCathodeMainPnP1AxisZ.commands.enableAxis := FALSE;
       "Unit1.Em5.HmiInterface".cmCathodeMainPnP1AxisZ.commands.enableAxis := TRUE;
   END_IF;
   IF #_w11 AND "Unit1.Em5.ControlNodes".cmCathodeMainPnP2AxisZ.monitoring.axisEnabled THEN
       "Unit1.Em5.ControlNodes".cmCathodeMainPnP2AxisZ.commands.enableAxis := FALSE;
       "Unit1.Em5.HmiInterface".cmCathodeMainPnP2AxisZ.commands.enableAxis := TRUE;
   END_IF;
   IF #_w11 AND "Unit1.Em5.ControlNodes".cmCathodeAlignTableAxisX.monitoring.axisEnabled THEN
       "Unit1.Em5.ControlNodes".cmCathodeAlignTableAxisX.commands.enableAxis := FALSE;
       "Unit1.Em5.HmiInterface".cmCathodeAlignTableAxisX.commands.enableAxis := TRUE;
   END_IF;
   IF #_w11 AND "Unit1.Em5.ControlNodes".cmCathodeAlignTableAxisY1.monitoring.axisEnabled THEN
       "Unit1.Em5.ControlNodes".cmCathodeAlignTableAxisY1.commands.enableAxis := FALSE;
       "Unit1.Em5.HmiInterface".cmCathodeAlignTableAxisY1.commands.enableAxis := TRUE;
   END_IF;
   IF #_w11 AND "Unit1.Em5.ControlNodes".cmCathodeAlignTableAxisY2.monitoring.axisEnabled THEN
       "Unit1.Em5.ControlNodes".cmCathodeAlignTableAxisY2.commands.enableAxis := FALSE;
       "Unit1.Em5.HmiInterface".cmCathodeAlignTableAxisY2.commands.enableAxis := TRUE;
   END_IF;
END_REGION

REGION Network 75: PHMI Servo Enable CMs
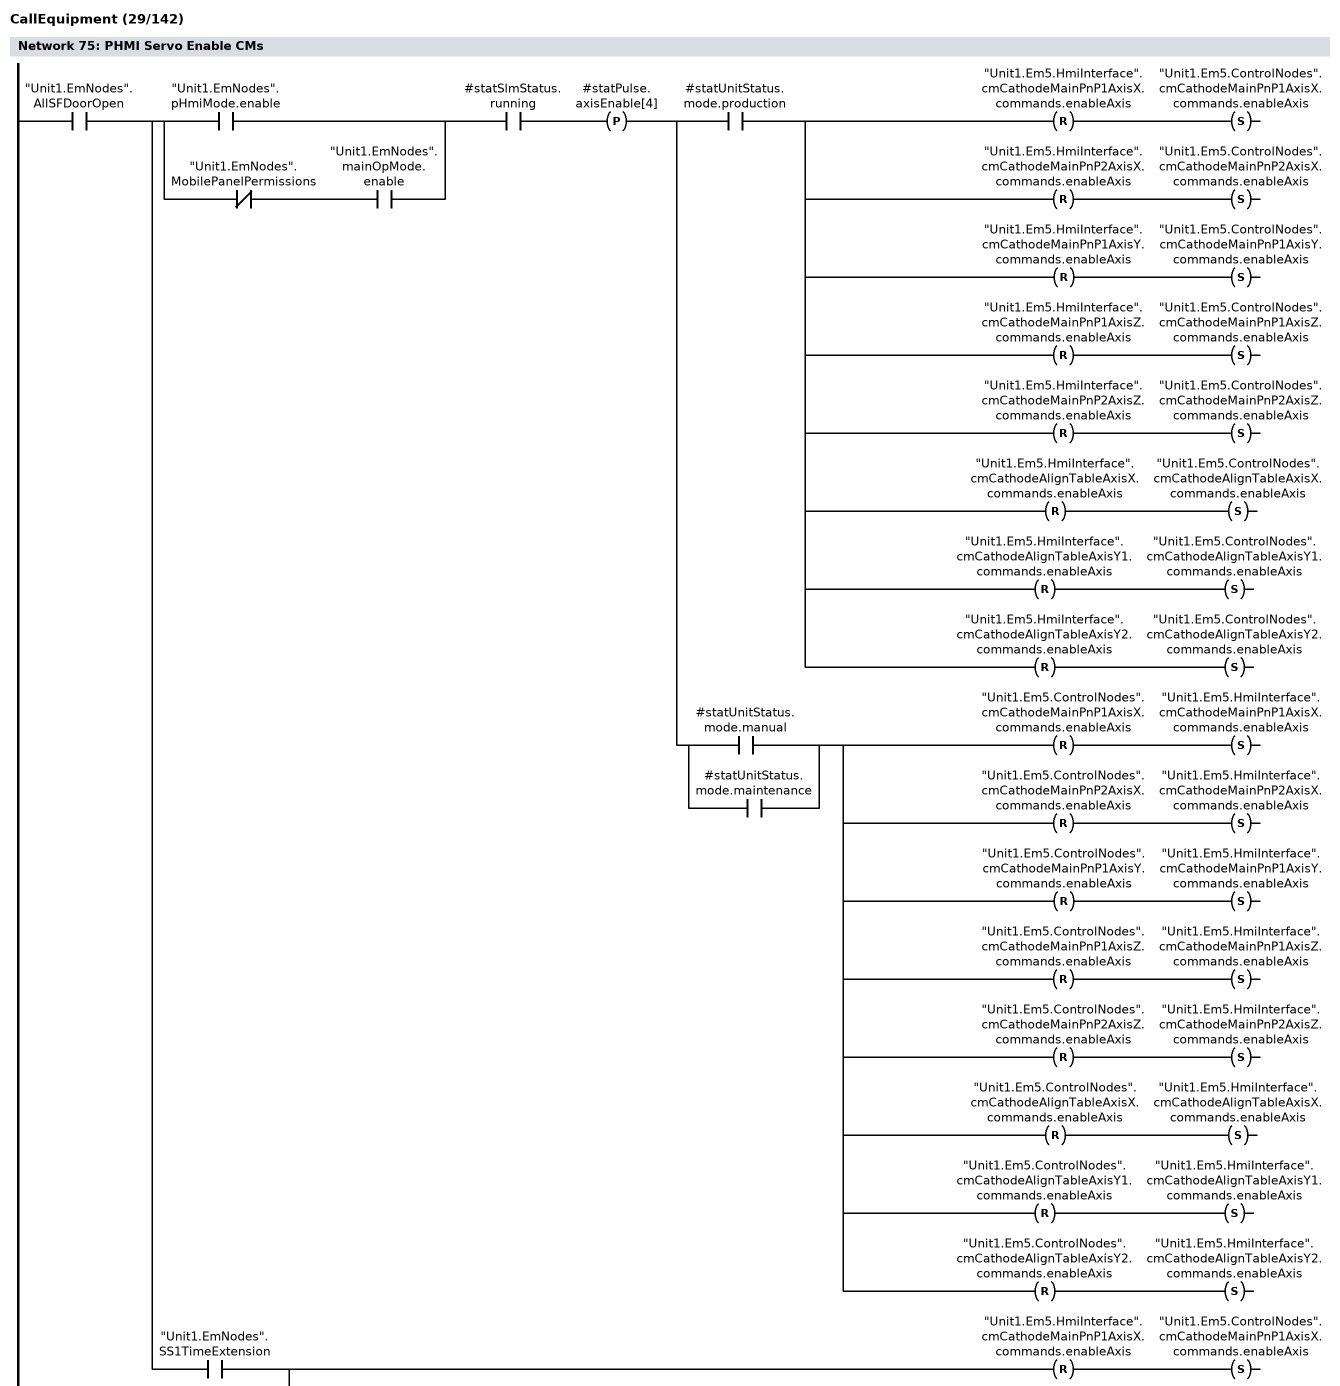
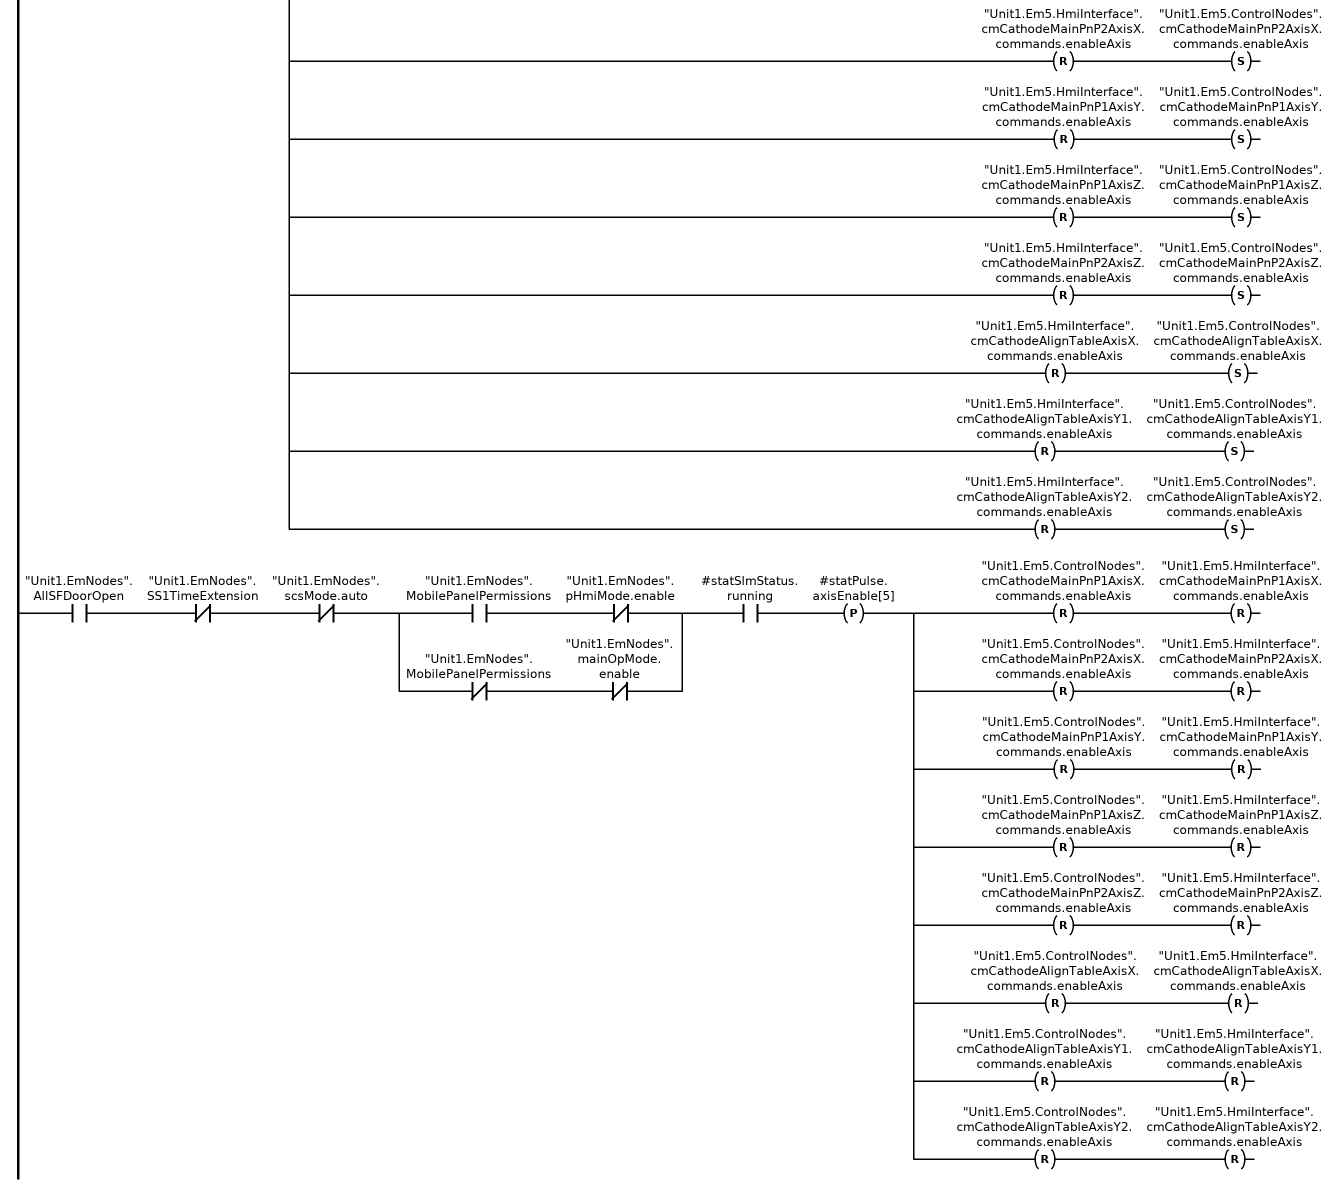
   RUNG wire#powerrail
      Contact( "Unit1.EmNodes".AllSFDoorOpen )
      wire#w1
      Contact( "Unit1.EmNodes".pHmiMode.enable )
      wire#w2
      Contact( #statSlmStatus.running )
      P_Trig( #statPulse.axisEnable[4] )
      wire#w3
      Contact( #statUnitStatus.mode.production )
      wire#w4
      R_Coil( "Unit1.Em5.HmiInterface".cmCathodeMainPnP1AxisX.commands.enableAxis )
      S_Coil( "Unit1.Em5.ControlNodes".cmCathodeMainPnP1AxisX.commands.enableAxis )
   END_RUNG
   RUNG wire#w1
      I_Contact( "Unit1.EmNodes".MobilePanelPermissions )
      Contact( "Unit1.EmNodes".mainOpMode.enable )
   END_RUNG wire#w2
   RUNG wire#w4
      R_Coil( "Unit1.Em5.HmiInterface".cmCathodeMainPnP2AxisX.commands.enableAxis )
      S_Coil( "Unit1.Em5.ControlNodes".cmCathodeMainPnP2AxisX.commands.enableAxis )
   END_RUNG
   RUNG wire#w4
      R_Coil( "Unit1.Em5.HmiInterface".cmCathodeMainPnP1AxisY.commands.enableAxis )
      S_Coil( "Unit1.Em5.ControlNodes".cmCathodeMainPnP1AxisY.commands.enableAxis )
   END_RUNG
   RUNG wire#w4
      R_Coil( "Unit1.Em5.HmiInterface".cmCathodeMainPnP1AxisZ.commands.enableAxis )
      S_Coil( "Unit1.Em5.ControlNodes".cmCathodeMainPnP1AxisZ.commands.enableAxis )
   END_RUNG
   RUNG wire#w4
      R_Coil( "Unit1.Em5.HmiInterface".cmCathodeMainPnP2AxisZ.commands.enableAxis )
      S_Coil( "Unit1.Em5.ControlNodes".cmCathodeMainPnP2AxisZ.commands.enableAxis )
   END_RUNG
   RUNG wire#w4
      R_Coil( "Unit1.Em5.HmiInterface".cmCathodeAlignTableAxisX.commands.enableAxis )
      S_Coil( "Unit1.Em5.ControlNodes".cmCathodeAlignTableAxisX.commands.enableAxis )
   END_RUNG
   RUNG wire#w4
      R_Coil( "Unit1.Em5.HmiInterface".cmCathodeAlignTableAxisY1.commands.enableAxis )
      S_Coil( "Unit1.Em5.ControlNodes".cmCathodeAlignTableAxisY1.commands.enableAxis )
   END_RUNG
   RUNG wire#w4
      R_Coil( "Unit1.Em5.HmiInterface".cmCathodeAlignTableAxisY2.commands.enableAxis )
      S_Coil( "Unit1.Em5.ControlNodes".cmCathodeAlignTableAxisY2.commands.enableAxis )
   END_RUNG
   RUNG wire#w3
      Contact( #statUnitStatus.mode.manual )
      wire#w5
      R_Coil( "Unit1.Em5.ControlNodes".cmCathodeMainPnP1AxisX.commands.enableAxis )
      S_Coil( "Unit1.Em5.HmiInterface".cmCathodeMainPnP1AxisX.commands.enableAxis )
   END_RUNG
   RUNG wire#w3
      Contact( #statUnitStatus.mode.maintenance )
   END_RUNG wire#w5
   RUNG wire#w5
      R_Coil( "Unit1.Em5.ControlNodes".cmCathodeMainPnP2AxisX.commands.enableAxis )
      S_Coil( "Unit1.Em5.HmiInterface".cmCathodeMainPnP2AxisX.commands.enableAxis )
   END_RUNG
   RUNG wire#w5
      R_Coil( "Unit1.Em5.ControlNodes".cmCathodeMainPnP1AxisY.commands.enableAxis )
      S_Coil( "Unit1.Em5.HmiInterface".cmCathodeMainPnP1AxisY.commands.enableAxis )
   END_RUNG
   RUNG wire#w5
      R_Coil( "Unit1.Em5.ControlNodes".cmCathodeMainPnP1AxisZ.commands.enableAxis )
      S_Coil( "Unit1.Em5.HmiInterface".cmCathodeMainPnP1AxisZ.commands.enableAxis )
   END_RUNG
   RUNG wire#w5
      R_Coil( "Unit1.Em5.ControlNodes".cmCathodeMainPnP2AxisZ.commands.enableAxis )
      S_Coil( "Unit1.Em5.HmiInterface".cmCathodeMainPnP2AxisZ.commands.enableAxis )
   END_RUNG
   RUNG wire#w5
      R_Coil( "Unit1.Em5.ControlNodes".cmCathodeAlignTableAxisX.commands.enableAxis )
      S_Coil( "Unit1.Em5.HmiInterface".cmCathodeAlignTableAxisX.commands.enableAxis )
   END_RUNG
   RUNG wire#w5
      R_Coil( "Unit1.Em5.ControlNodes".cmCathodeAlignTableAxisY1.commands.enableAxis )
      S_Coil( "Unit1.Em5.HmiInterface".cmCathodeAlignTableAxisY1.commands.enableAxis )
   END_RUNG
   RUNG wire#w5
      R_Coil( "Unit1.Em5.ControlNodes".cmCathodeAlignTableAxisY2.commands.enableAxis )
      S_Coil( "Unit1.Em5.HmiInterface".cmCathodeAlignTableAxisY2.commands.enableAxis )
   END_RUNG
   RUNG wire#w1
      Contact( "Unit1.EmNodes".SS1TimeExtension )
      wire#w6
      R_Coil( "Unit1.Em5.HmiInterface".cmCathodeMainPnP1AxisX.commands.enableAxis )
      S_Coil( "Unit1.Em5.ControlNodes".cmCathodeMainPnP1AxisX.commands.enableAxis )
   END_RUNG
   RUNG wire#w6
      R_Coil( "Unit1.Em5.HmiInterface".cmCathodeMainPnP2AxisX.commands.enableAxis )
      S_Coil( "Unit1.Em5.ControlNodes".cmCathodeMainPnP2AxisX.commands.enableAxis )
   END_RUNG
   RUNG wire#w6
      R_Coil( "Unit1.Em5.HmiInterface".cmCathodeMainPnP1AxisY.commands.enableAxis )
      S_Coil( "Unit1.Em5.ControlNodes".cmCathodeMainPnP1AxisY.commands.enableAxis )
   END_RUNG
   RUNG wire#w6
      R_Coil( "Unit1.Em5.HmiInterface".cmCathodeMainPnP1AxisZ.commands.enableAxis )
      S_Coil( "Unit1.Em5.ControlNodes".cmCathodeMainPnP1AxisZ.commands.enableAxis )
   END_RUNG
   RUNG wire#w6
      R_Coil( "Unit1.Em5.HmiInterface".cmCathodeMainPnP2AxisZ.commands.enableAxis )
      S_Coil( "Unit1.Em5.ControlNodes".cmCathodeMainPnP2AxisZ.commands.enableAxis )
   END_RUNG
   RUNG wire#w6
      R_Coil( "Unit1.Em5.HmiInterface".cmCathodeAlignTableAxisX.commands.enableAxis )
      S_Coil( "Unit1.Em5.ControlNodes".cmCathodeAlignTableAxisX.commands.enableAxis )
   END_RUNG
   RUNG wire#w6
      R_Coil( "Unit1.Em5.HmiInterface".cmCathodeAlignTableAxisY1.commands.enableAxis )
      S_Coil( "Unit1.Em5.ControlNodes".cmCathodeAlignTableAxisY1.commands.enableAxis )
   END_RUNG
   RUNG wire#w6
      R_Coil( "Unit1.Em5.HmiInterface".cmCathodeAlignTableAxisY2.commands.enableAxis )
      S_Coil( "Unit1.Em5.ControlNodes".cmCathodeAlignTableAxisY2.commands.enableAxis )
   END_RUNG
   RUNG wire#powerrail
      Contact( "Unit1.EmNodes".AllSFDoorOpen )
      I_Contact( "Unit1.EmNodes".SS1TimeExtension )
      I_Contact( "Unit1.EmNodes".scsMode.auto )
      wire#w7
      Contact( "Unit1.EmNodes".MobilePanelPermissions )
      I_Contact( "Unit1.EmNodes".pHmiMode.enable )
      wire#w8
      Contact( #statSlmStatus.running )
      P_Trig( #statPulse.axisEnable[5] )
      wire#w9
      R_Coil( "Unit1.Em5.ControlNodes".cmCathodeMainPnP1AxisX.commands.enableAxis )
      R_Coil( "Unit1.Em5.HmiInterface".cmCathodeMainPnP1AxisX.commands.enableAxis )
   END_RUNG
   RUNG wire#w7
      I_Contact( "Unit1.EmNodes".MobilePanelPermissions )
      I_Contact( "Unit1.EmNodes".mainOpMode.enable )
   END_RUNG wire#w8
   RUNG wire#w9
      R_Coil( "Unit1.Em5.ControlNodes".cmCathodeMainPnP2AxisX.commands.enableAxis )
      R_Coil( "Unit1.Em5.HmiInterface".cmCathodeMainPnP2AxisX.commands.enableAxis )
   END_RUNG
   RUNG wire#w9
      R_Coil( "Unit1.Em5.ControlNodes".cmCathodeMainPnP1AxisY.commands.enableAxis )
      R_Coil( "Unit1.Em5.HmiInterface".cmCathodeMainPnP1AxisY.commands.enableAxis )
   END_RUNG
   RUNG wire#w9
      R_Coil( "Unit1.Em5.ControlNodes".cmCathodeMainPnP1AxisZ.commands.enableAxis )
      R_Coil( "Unit1.Em5.HmiInterface".cmCathodeMainPnP1AxisZ.commands.enableAxis )
   END_RUNG
   RUNG wire#w9
      R_Coil( "Unit1.Em5.ControlNodes".cmCathodeMainPnP2AxisZ.commands.enableAxis )
      R_Coil( "Unit1.Em5.HmiInterface".cmCathodeMainPnP2AxisZ.commands.enableAxis )
   END_RUNG
   RUNG wire#w9
      R_Coil( "Unit1.Em5.ControlNodes".cmCathodeAlignTableAxisX.commands.enableAxis )
      R_Coil( "Unit1.Em5.HmiInterface".cmCathodeAlignTableAxisX.commands.enableAxis )
   END_RUNG
   RUNG wire#w9
      R_Coil( "Unit1.Em5.ControlNodes".cmCathodeAlignTableAxisY1.commands.enableAxis )
      R_Coil( "Unit1.Em5.HmiInterface".cmCathodeAlignTableAxisY1.commands.enableAxis )
   END_RUNG
   RUNG wire#w9
      R_Coil( "Unit1.Em5.ControlNodes".cmCathodeAlignTableAxisY2.commands.enableAxis )
      R_Coil( "Unit1.Em5.HmiInterface".cmCathodeAlignTableAxisY2.commands.enableAxis )
   END_RUNG
   // the same network as SCL:
   #_w1 := "Unit1.EmNodes".AllSFDoorOpen AND ("Unit1.EmNodes".pHmiMode.enable OR (NOT "Unit1.EmNodes".MobilePanelPermissions AND "Unit1.EmNodes".mainOpMode.enable)) AND #statSlmStatus.running;
   #_w2 := #_w1 AND NOT #statPulse.axisEnable[4];   // rising edge
   #statPulse.axisEnable[4] := #_w1;
   IF #_w2 AND #statUnitStatus.mode.production THEN
       "Unit1.Em5.HmiInterface".cmCathodeMainPnP1AxisX.commands.enableAxis := FALSE;
       "Unit1.Em5.ControlNodes".cmCathodeMainPnP1AxisX.commands.enableAxis := TRUE;
       "Unit1.Em5.HmiInterface".cmCathodeMainPnP2AxisX.commands.enableAxis := FALSE;
       "Unit1.Em5.ControlNodes".cmCathodeMainPnP2AxisX.commands.enableAxis := TRUE;
       "Unit1.Em5.HmiInterface".cmCathodeMainPnP1AxisY.commands.enableAxis := FALSE;
       "Unit1.Em5.ControlNodes".cmCathodeMainPnP1AxisY.commands.enableAxis := TRUE;
       "Unit1.Em5.HmiInterface".cmCathodeMainPnP1AxisZ.commands.enableAxis := FALSE;
       "Unit1.Em5.ControlNodes".cmCathodeMainPnP1AxisZ.commands.enableAxis := TRUE;
       "Unit1.Em5.HmiInterface".cmCathodeMainPnP2AxisZ.commands.enableAxis := FALSE;
       "Unit1.Em5.ControlNodes".cmCathodeMainPnP2AxisZ.commands.enableAxis := TRUE;
       "Unit1.Em5.HmiInterface".cmCathodeAlignTableAxisX.commands.enableAxis := FALSE;
       "Unit1.Em5.ControlNodes".cmCathodeAlignTableAxisX.commands.enableAxis := TRUE;
       "Unit1.Em5.HmiInterface".cmCathodeAlignTableAxisY1.commands.enableAxis := FALSE;
       "Unit1.Em5.ControlNodes".cmCathodeAlignTableAxisY1.commands.enableAxis := TRUE;
       "Unit1.Em5.HmiInterface".cmCathodeAlignTableAxisY2.commands.enableAxis := FALSE;
       "Unit1.Em5.ControlNodes".cmCathodeAlignTableAxisY2.commands.enableAxis := TRUE;
   END_IF;
   IF #_w2 AND (#statUnitStatus.mode.manual OR #statUnitStatus.mode.maintenance) THEN
       "Unit1.Em5.ControlNodes".cmCathodeMainPnP1AxisX.commands.enableAxis := FALSE;
       "Unit1.Em5.HmiInterface".cmCathodeMainPnP1AxisX.commands.enableAxis := TRUE;
       "Unit1.Em5.ControlNodes".cmCathodeMainPnP2AxisX.commands.enableAxis := FALSE;
       "Unit1.Em5.HmiInterface".cmCathodeMainPnP2AxisX.commands.enableAxis := TRUE;
       "Unit1.Em5.ControlNodes".cmCathodeMainPnP1AxisY.commands.enableAxis := FALSE;
       "Unit1.Em5.HmiInterface".cmCathodeMainPnP1AxisY.commands.enableAxis := TRUE;
       "Unit1.Em5.ControlNodes".cmCathodeMainPnP1AxisZ.commands.enableAxis := FALSE;
       "Unit1.Em5.HmiInterface".cmCathodeMainPnP1AxisZ.commands.enableAxis := TRUE;
       "Unit1.Em5.ControlNodes".cmCathodeMainPnP2AxisZ.commands.enableAxis := FALSE;
       "Unit1.Em5.HmiInterface".cmCathodeMainPnP2AxisZ.commands.enableAxis := TRUE;
       "Unit1.Em5.ControlNodes".cmCathodeAlignTableAxisX.commands.enableAxis := FALSE;
       "Unit1.Em5.HmiInterface".cmCathodeAlignTableAxisX.commands.enableAxis := TRUE;
       "Unit1.Em5.ControlNodes".cmCathodeAlignTableAxisY1.commands.enableAxis := FALSE;
       "Unit1.Em5.HmiInterface".cmCathodeAlignTableAxisY1.commands.enableAxis := TRUE;
       "Unit1.Em5.ControlNodes".cmCathodeAlignTableAxisY2.commands.enableAxis := FALSE;
       "Unit1.Em5.HmiInterface".cmCathodeAlignTableAxisY2.commands.enableAxis := TRUE;
   END_IF;
   IF "Unit1.EmNodes".AllSFDoorOpen AND "Unit1.EmNodes".SS1TimeExtension THEN
       "Unit1.Em5.HmiInterface".cmCathodeMainPnP1AxisX.commands.enableAxis := FALSE;
       "Unit1.Em5.ControlNodes".cmCathodeMainPnP1AxisX.commands.enableAxis := TRUE;
       "Unit1.Em5.HmiInterface".cmCathodeMainPnP2AxisX.commands.enableAxis := FALSE;
       "Unit1.Em5.ControlNodes".cmCathodeMainPnP2AxisX.commands.enableAxis := TRUE;
       "Unit1.Em5.HmiInterface".cmCathodeMainPnP1AxisY.commands.enableAxis := FALSE;
       "Unit1.Em5.ControlNodes".cmCathodeMainPnP1AxisY.commands.enableAxis := TRUE;
       "Unit1.Em5.HmiInterface".cmCathodeMainPnP1AxisZ.commands.enableAxis := FALSE;
       "Unit1.Em5.ControlNodes".cmCathodeMainPnP1AxisZ.commands.enableAxis := TRUE;
       "Unit1.Em5.HmiInterface".cmCathodeMainPnP2AxisZ.commands.enableAxis := FALSE;
       "Unit1.Em5.ControlNodes".cmCathodeMainPnP2AxisZ.commands.enableAxis := TRUE;
       "Unit1.Em5.HmiInterface".cmCathodeAlignTableAxisX.commands.enableAxis := FALSE;
       "Unit1.Em5.ControlNodes".cmCathodeAlignTableAxisX.commands.enableAxis := TRUE;
       "Unit1.Em5.HmiInterface".cmCathodeAlignTableAxisY1.commands.enableAxis := FALSE;
       "Unit1.Em5.ControlNodes".cmCathodeAlignTableAxisY1.commands.enableAxis := TRUE;
       "Unit1.Em5.HmiInterface".cmCathodeAlignTableAxisY2.commands.enableAxis := FALSE;
       "Unit1.Em5.ControlNodes".cmCathodeAlignTableAxisY2.commands.enableAxis := TRUE;
   END_IF;
   #_w3 := "Unit1.EmNodes".AllSFDoorOpen AND NOT "Unit1.EmNodes".SS1TimeExtension AND NOT "Unit1.EmNodes".scsMode.auto AND (("Unit1.EmNodes".MobilePanelPermissions AND NOT "Unit1.EmNodes".pHmiMode.enable) OR (NOT "Unit1.EmNodes".MobilePanelPermissions AND NOT "Unit1.EmNodes".mainOpMode.enable)) AND #statSlmStatus.running;
   #_w4 := #_w3 AND NOT #statPulse.axisEnable[5];   // rising edge
   #statPulse.axisEnable[5] := #_w3;
   IF #_w4 THEN
       "Unit1.Em5.ControlNodes".cmCathodeMainPnP1AxisX.commands.enableAxis := FALSE;
       "Unit1.Em5.HmiInterface".cmCathodeMainPnP1AxisX.commands.enableAxis := FALSE;
       "Unit1.Em5.ControlNodes".cmCathodeMainPnP2AxisX.commands.enableAxis := FALSE;
       "Unit1.Em5.HmiInterface".cmCathodeMainPnP2AxisX.commands.enableAxis := FALSE;
       "Unit1.Em5.ControlNodes".cmCathodeMainPnP1AxisY.commands.enableAxis := FALSE;
       "Unit1.Em5.HmiInterface".cmCathodeMainPnP1AxisY.commands.enableAxis := FALSE;
       "Unit1.Em5.ControlNodes".cmCathodeMainPnP1AxisZ.commands.enableAxis := FALSE;
       "Unit1.Em5.HmiInterface".cmCathodeMainPnP1AxisZ.commands.enableAxis := FALSE;
       "Unit1.Em5.ControlNodes".cmCathodeMainPnP2AxisZ.commands.enableAxis := FALSE;
       "Unit1.Em5.HmiInterface".cmCathodeMainPnP2AxisZ.commands.enableAxis := FALSE;
       "Unit1.Em5.ControlNodes".cmCathodeAlignTableAxisX.commands.enableAxis := FALSE;
       "Unit1.Em5.HmiInterface".cmCathodeAlignTableAxisX.commands.enableAxis := FALSE;
       "Unit1.Em5.ControlNodes".cmCathodeAlignTableAxisY1.commands.enableAxis := FALSE;
       "Unit1.Em5.HmiInterface".cmCathodeAlignTableAxisY1.commands.enableAxis := FALSE;
       "Unit1.Em5.ControlNodes".cmCathodeAlignTableAxisY2.commands.enableAxis := FALSE;
       "Unit1.Em5.HmiInterface".cmCathodeAlignTableAxisY2.commands.enableAxis := FALSE;
   END_IF;
END_REGION

REGION Network 76: Disable All CMs
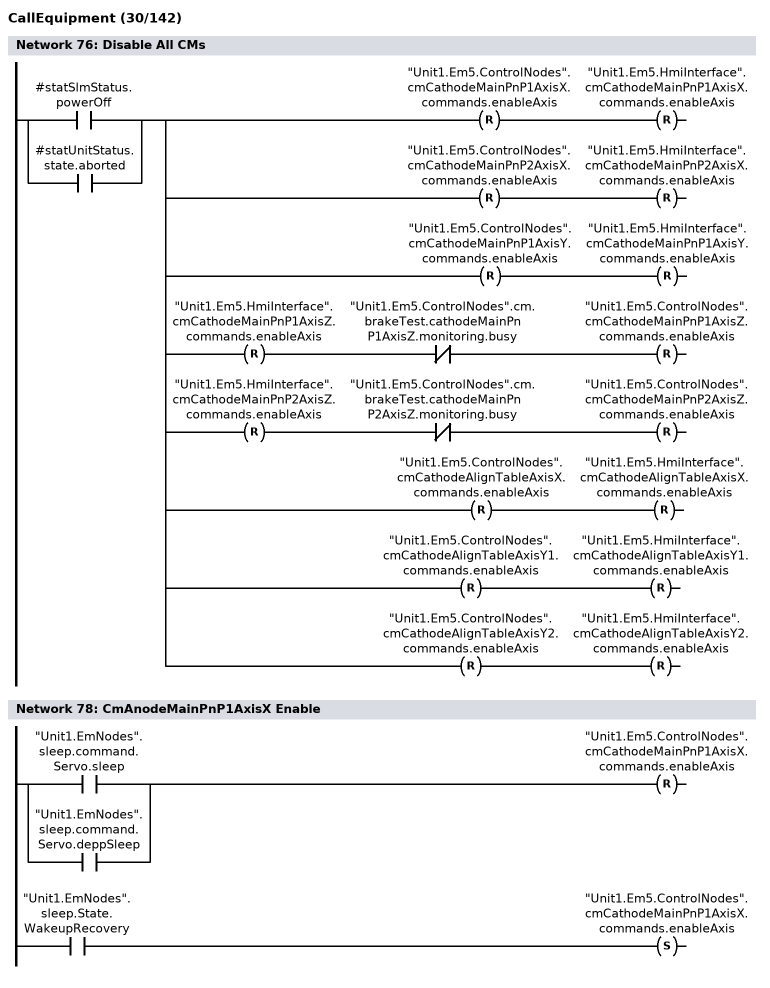
   RUNG wire#powerrail
      Contact( #statSlmStatus.powerOff )
      wire#w1
      R_Coil( "Unit1.Em5.ControlNodes".cmCathodeMainPnP1AxisX.commands.enableAxis )
      R_Coil( "Unit1.Em5.HmiInterface".cmCathodeMainPnP1AxisX.commands.enableAxis )
   END_RUNG
   RUNG wire#powerrail
      Contact( #statUnitStatus.state.aborted )
   END_RUNG wire#w1
   RUNG wire#w1
      R_Coil( "Unit1.Em5.ControlNodes".cmCathodeMainPnP2AxisX.commands.enableAxis )
      R_Coil( "Unit1.Em5.HmiInterface".cmCathodeMainPnP2AxisX.commands.enableAxis )
   END_RUNG
   RUNG wire#w1
      R_Coil( "Unit1.Em5.ControlNodes".cmCathodeMainPnP1AxisY.commands.enableAxis )
      R_Coil( "Unit1.Em5.HmiInterface".cmCathodeMainPnP1AxisY.commands.enableAxis )
   END_RUNG
   RUNG wire#w1
      R_Coil( "Unit1.Em5.HmiInterface".cmCathodeMainPnP1AxisZ.commands.enableAxis )
      I_Contact( "Unit1.Em5.ControlNodes".cm.brakeTest.cathodeMainPnP1AxisZ.monitoring.busy )
      R_Coil( "Unit1.Em5.ControlNodes".cmCathodeMainPnP1AxisZ.commands.enableAxis )
   END_RUNG
   RUNG wire#w1
      R_Coil( "Unit1.Em5.HmiInterface".cmCathodeMainPnP2AxisZ.commands.enableAxis )
      I_Contact( "Unit1.Em5.ControlNodes".cm.brakeTest.cathodeMainPnP2AxisZ.monitoring.busy )
      R_Coil( "Unit1.Em5.ControlNodes".cmCathodeMainPnP2AxisZ.commands.enableAxis )
   END_RUNG
   RUNG wire#w1
      R_Coil( "Unit1.Em5.ControlNodes".cmCathodeAlignTableAxisX.commands.enableAxis )
      R_Coil( "Unit1.Em5.HmiInterface".cmCathodeAlignTableAxisX.commands.enableAxis )
   END_RUNG
   RUNG wire#w1
      R_Coil( "Unit1.Em5.ControlNodes".cmCathodeAlignTableAxisY1.commands.enableAxis )
      R_Coil( "Unit1.Em5.HmiInterface".cmCathodeAlignTableAxisY1.commands.enableAxis )
   END_RUNG
   RUNG wire#w1
      R_Coil( "Unit1.Em5.ControlNodes".cmCathodeAlignTableAxisY2.commands.enableAxis )
      R_Coil( "Unit1.Em5.HmiInterface".cmCathodeAlignTableAxisY2.commands.enableAxis )
   END_RUNG
   // the same network as SCL:
   #_w1 := #statSlmStatus.powerOff OR #statUnitStatus.state.aborted;
   IF #_w1 THEN
       "Unit1.Em5.ControlNodes".cmCathodeMainPnP1AxisX.commands.enableAxis := FALSE;
       "Unit1.Em5.HmiInterface".cmCathodeMainPnP1AxisX.commands.enableAxis := FALSE;
       "Unit1.Em5.ControlNodes".cmCathodeMainPnP2AxisX.commands.enableAxis := FALSE;
       "Unit1.Em5.HmiInterface".cmCathodeMainPnP2AxisX.commands.enableAxis := FALSE;
       "Unit1.Em5.ControlNodes".cmCathodeMainPnP1AxisY.commands.enableAxis := FALSE;
       "Unit1.Em5.HmiInterface".cmCathodeMainPnP1AxisY.commands.enableAxis := FALSE;
       "Unit1.Em5.HmiInterface".cmCathodeMainPnP1AxisZ.commands.enableAxis := FALSE;
   END_IF;
   IF #_w1 AND NOT "Unit1.Em5.ControlNodes".cm.brakeTest.cathodeMainPnP1AxisZ.monitoring.busy THEN
       "Unit1.Em5.ControlNodes".cmCathodeMainPnP1AxisZ.commands.enableAxis := FALSE;
   END_IF;
   IF #_w1 THEN "Unit1.Em5.HmiInterface".cmCathodeMainPnP2AxisZ.commands.enableAxis := FALSE; END_IF;
   IF #_w1 AND NOT "Unit1.Em5.ControlNodes".cm.brakeTest.cathodeMainPnP2AxisZ.monitoring.busy THEN
       "Unit1.Em5.ControlNodes".cmCathodeMainPnP2AxisZ.commands.enableAxis := FALSE;
   END_IF;
   IF #_w1 THEN
       "Unit1.Em5.ControlNodes".cmCathodeAlignTableAxisX.commands.enableAxis := FALSE;
       "Unit1.Em5.HmiInterface".cmCathodeAlignTableAxisX.commands.enableAxis := FALSE;
       "Unit1.Em5.ControlNodes".cmCathodeAlignTableAxisY1.commands.enableAxis := FALSE;
       "Unit1.Em5.HmiInterface".cmCathodeAlignTableAxisY1.commands.enableAxis := FALSE;
       "Unit1.Em5.ControlNodes".cmCathodeAlignTableAxisY2.commands.enableAxis := FALSE;
       "Unit1.Em5.HmiInterface".cmCathodeAlignTableAxisY2.commands.enableAxis := FALSE;
   END_IF;
END_REGION

REGION Network 78: CmAnodeMainPnP1AxisX Enable
   RUNG wire#powerrail
      Contact( "Unit1.EmNodes".sleep.command.Servo.sleep )
      wire#w1
      R_Coil( "Unit1.Em5.ControlNodes".cmCathodeMainPnP1AxisX.commands.enableAxis )
   END_RUNG
   RUNG wire#powerrail
      Contact( "Unit1.EmNodes".sleep.command.Servo.deppSleep )
   END_RUNG wire#w1
   RUNG wire#powerrail
      Contact( "Unit1.EmNodes".sleep.State.WakeupRecovery )
      S_Coil( "Unit1.Em5.ControlNodes".cmCathodeMainPnP1AxisX.commands.enableAxis )
   END_RUNG
   // the same network as SCL:
   IF "Unit1.EmNodes".sleep.command.Servo.sleep OR "Unit1.EmNodes".sleep.command.Servo.deppSleep THEN
       "Unit1.Em5.ControlNodes".cmCathodeMainPnP1AxisX.commands.enableAxis := FALSE;
   END_IF;
   IF "Unit1.EmNodes".sleep.State.WakeupRecovery THEN
       "Unit1.Em5.ControlNodes".cmCathodeMainPnP1AxisX.commands.enableAxis := TRUE;
   END_IF;
END_REGION

REGION Network 79: cathode Main P&P 1 X-Axis Homing Interlock
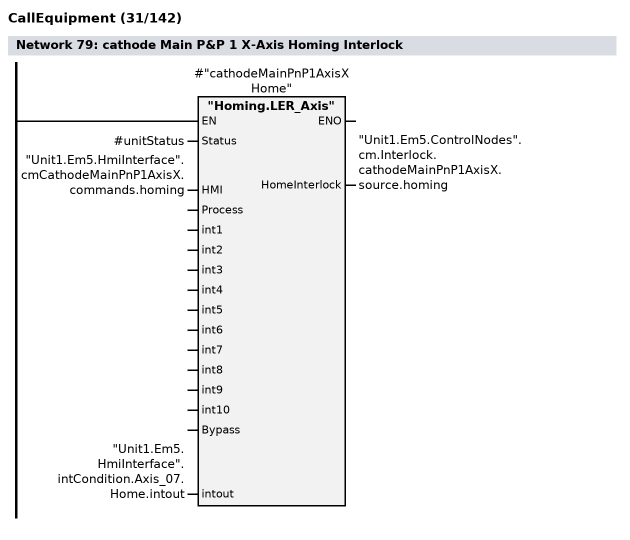
   RUNG wire#powerrail
      #"cathodeMainPnP1AxisX Home"(Status := #unitStatus, HMI := "Unit1.Em5.HmiInterface".cmCathodeMainPnP1AxisX.commands.homing, Process :=, int1 :=, int2 :=, int3 :=, int4 :=, int5 :=, int6 :=, int7 :=, int8 :=, int9 :=, int10 :=, Bypass :=, intout := "Unit1.Em5.HmiInterface".intCondition.Axis_07.Home.intout, HomeInterlock => "Unit1.Em5.ControlNodes".cm.Interlock.cathodeMainPnP1AxisX.source.homing)
   END_RUNG
   // the same network as SCL:
   #"cathodeMainPnP1AxisX Home"(Status := #unitStatus,   // "Homing.LER_Axis"
                           HMI := "Unit1.Em5.HmiInterface".cmCathodeMainPnP1AxisX.commands.homing,
                           intout := "Unit1.Em5.HmiInterface".intCondition.Axis_07.Home.intout,
                           HomeInterlock => "Unit1.Em5.ControlNodes".cm.Interlock.cathodeMainPnP1AxisX.source.homing);
END_REGION

REGION Network 80: CmCathodeMainPnP1AxisX Position Absolute Jog
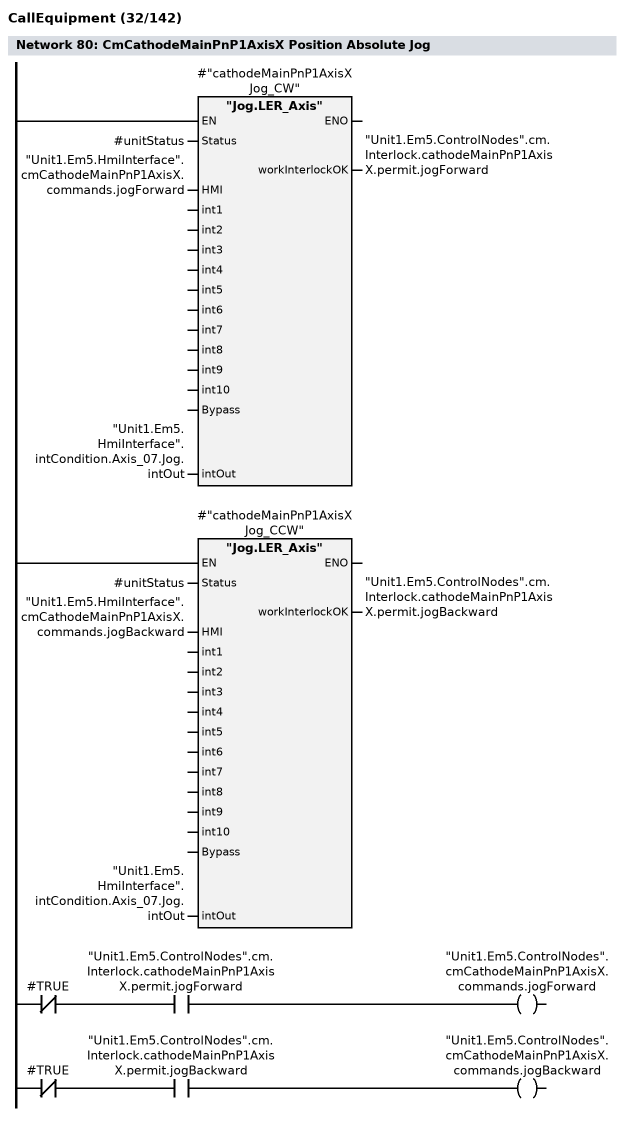
   RUNG wire#powerrail
      #"cathodeMainPnP1AxisX Jog_CW"(Status := #unitStatus, HMI := "Unit1.Em5.HmiInterface".cmCathodeMainPnP1AxisX.commands.jogForward, int1 :=, int2 :=, int3 :=, int4 :=, int5 :=, int6 :=, int7 :=, int8 :=, int9 :=, int10 :=, Bypass :=, intOut := "Unit1.Em5.HmiInterface".intCondition.Axis_07.Jog.intOut, workInterlockOK => "Unit1.Em5.ControlNodes".cm.Interlock.cathodeMainPnP1AxisX.permit.jogForward)
   END_RUNG
   RUNG wire#powerrail
      #"cathodeMainPnP1AxisX Jog_CCW"(Status := #unitStatus, HMI := "Unit1.Em5.HmiInterface".cmCathodeMainPnP1AxisX.commands.jogBackward, int1 :=, int2 :=, int3 :=, int4 :=, int5 :=, int6 :=, int7 :=, int8 :=, int9 :=, int10 :=, Bypass :=, intOut := "Unit1.Em5.HmiInterface".intCondition.Axis_07.Jog.intOut, workInterlockOK => "Unit1.Em5.ControlNodes".cm.Interlock.cathodeMainPnP1AxisX.permit.jogBackward)
   END_RUNG
   RUNG wire#powerrail
      I_Contact( #TRUE )
      Contact( "Unit1.Em5.ControlNodes".cm.Interlock.cathodeMainPnP1AxisX.permit.jogForward )
      Coil( "Unit1.Em5.ControlNodes".cmCathodeMainPnP1AxisX.commands.jogForward )
   END_RUNG
   RUNG wire#powerrail
      I_Contact( #TRUE )
      Contact( "Unit1.Em5.ControlNodes".cm.Interlock.cathodeMainPnP1AxisX.permit.jogBackward )
      Coil( "Unit1.Em5.ControlNodes".cmCathodeMainPnP1AxisX.commands.jogBackward )
   END_RUNG
   // the same network as SCL:
   #"cathodeMainPnP1AxisX Jog_CW"(Status := #unitStatus,   // "Jog.LER_Axis"
                           HMI := "Unit1.Em5.HmiInterface".cmCathodeMainPnP1AxisX.commands.jogForward,
                           intOut := "Unit1.Em5.HmiInterface".intCondition.Axis_07.Jog.intOut,
                           workInterlockOK => "Unit1.Em5.ControlNodes".cm.Interlock.cathodeMainPnP1AxisX.permit.jogForward);
   #"cathodeMainPnP1AxisX Jog_CCW"(Status := #unitStatus,   // "Jog.LER_Axis"
                           HMI := "Unit1.Em5.HmiInterface".cmCathodeMainPnP1AxisX.commands.jogBackward,
                           intOut := "Unit1.Em5.HmiInterface".intCondition.Axis_07.Jog.intOut,
                           workInterlockOK => "Unit1.Em5.ControlNodes".cm.Interlock.cathodeMainPnP1AxisX.permit.jogBackward);
   "Unit1.Em5.ControlNodes".cmCathodeMainPnP1AxisX.commands.jogForward := NOT #TRUE AND "Unit1.Em5.ControlNodes".cm.Interlock.cathodeMainPnP1AxisX.permit.jogForward;
   "Unit1.Em5.ControlNodes".cmCathodeMainPnP1AxisX.commands.jogBackward := NOT #TRUE AND "Unit1.Em5.ControlNodes".cm.Interlock.cathodeMainPnP1AxisX.permit.jogBackward;
END_REGION

REGION Network 81: CmCathodeMainPnP1AxisX Position Absolute Position0
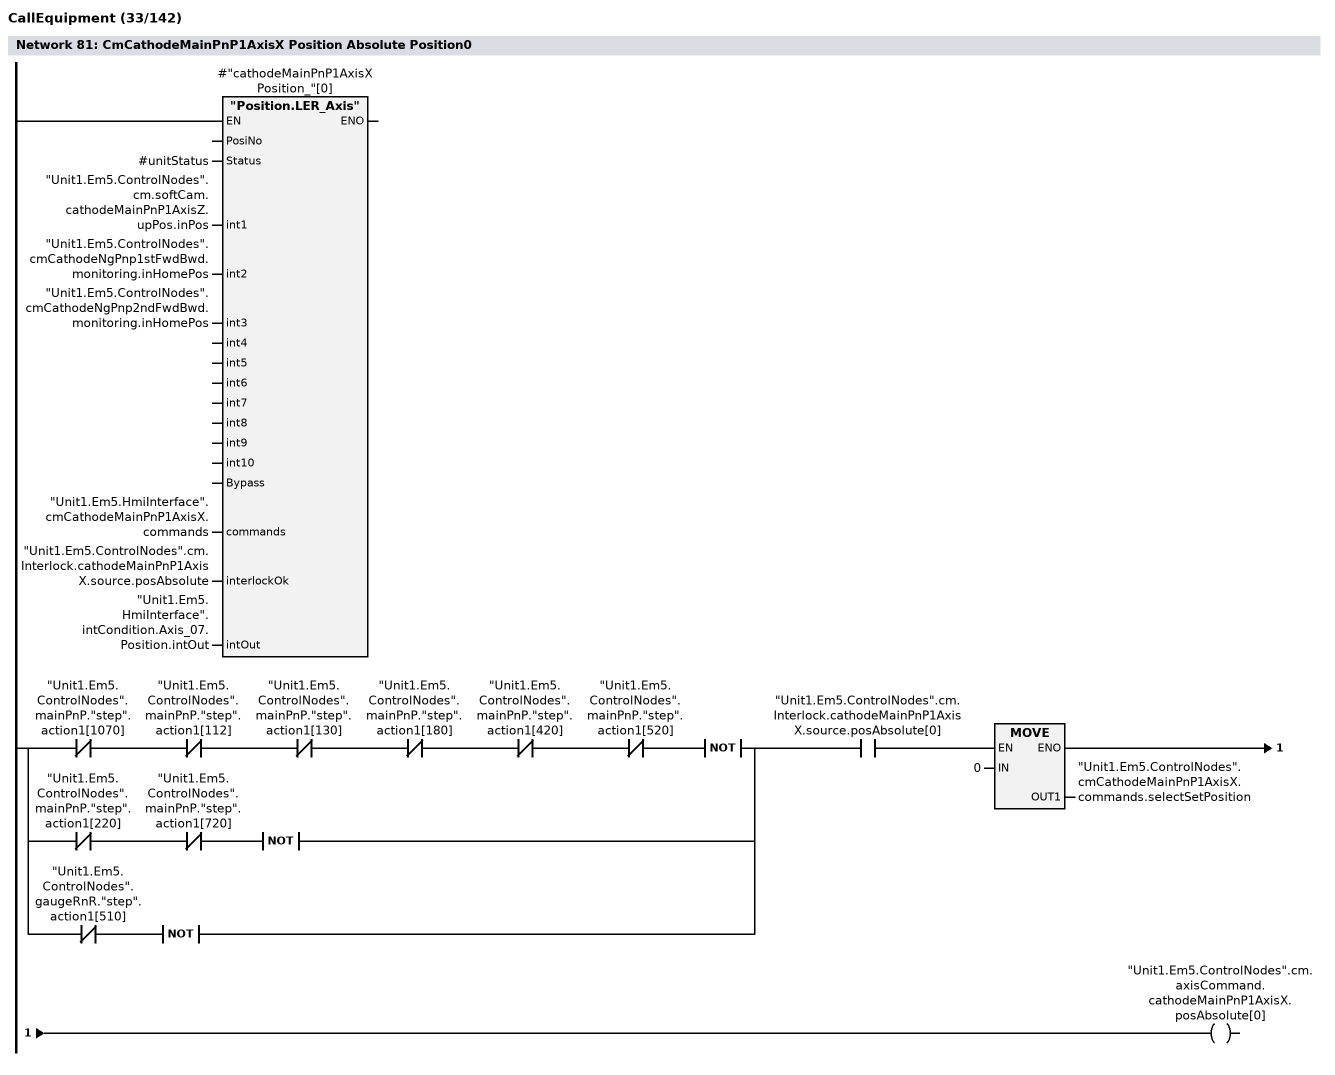
   RUNG wire#powerrail
      #"cathodeMainPnP1AxisX Position_"[0](PosiNo :=, Status := #unitStatus, int1 := "Unit1.Em5.ControlNodes".cm.softCam.cathodeMainPnP1AxisZ.upPos.inPos, int2 := "Unit1.Em5.ControlNodes".cmCathodeNgPnp1stFwdBwd.monitoring.inHomePos, int3 := "Unit1.Em5.ControlNodes".cmCathodeNgPnp2ndFwdBwd.monitoring.inHomePos, int4 :=, int5 :=, int6 :=, int7 :=, int8 :=, int9 :=, int10 :=, Bypass :=, commands := "Unit1.Em5.HmiInterface".cmCathodeMainPnP1AxisX.commands, interlockOk := "Unit1.Em5.ControlNodes".cm.Interlock.cathodeMainPnP1AxisX.source.posAbsolute, intOut := "Unit1.Em5.HmiInterface".intCondition.Axis_07.Position.intOut)
   END_RUNG
   RUNG wire#powerrail
      I_Contact( "Unit1.Em5.ControlNodes".mainPnP."step".action1[1070] )
      I_Contact( "Unit1.Em5.ControlNodes".mainPnP."step".action1[112] )
      I_Contact( "Unit1.Em5.ControlNodes".mainPnP."step".action1[130] )
      I_Contact( "Unit1.Em5.ControlNodes".mainPnP."step".action1[180] )
      I_Contact( "Unit1.Em5.ControlNodes".mainPnP."step".action1[420] )
      I_Contact( "Unit1.Em5.ControlNodes".mainPnP."step".action1[520] )
      Not()
      wire#w1
      Contact( "Unit1.Em5.ControlNodes".cm.Interlock.cathodeMainPnP1AxisX.source.posAbsolute[0] )
      Move(in := 0, out1 => "Unit1.Em5.ControlNodes".cmCathodeMainPnP1AxisX.commands.selectSetPosition)
      Coil( "Unit1.Em5.ControlNodes".cm.axisCommand.cathodeMainPnP1AxisX.posAbsolute[0] )
   END_RUNG
   RUNG wire#powerrail
      I_Contact( "Unit1.Em5.ControlNodes".mainPnP."step".action1[220] )
      I_Contact( "Unit1.Em5.ControlNodes".mainPnP."step".action1[720] )
      Not()
   END_RUNG wire#w1
   RUNG wire#powerrail
      I_Contact( "Unit1.Em5.ControlNodes".gaugeRnR."step".action1[510] )
      Not()
   END_RUNG wire#w1
   // the same network as SCL:
   #"cathodeMainPnP1AxisX Position_"[0](Status := #unitStatus,   // "Position.LER_Axis"
                           int1 := "Unit1.Em5.ControlNodes".cm.softCam.cathodeMainPnP1AxisZ.upPos.inPos,
                           int2 := "Unit1.Em5.ControlNodes".cmCathodeNgPnp1stFwdBwd.monitoring.inHomePos,
                           int3 := "Unit1.Em5.ControlNodes".cmCathodeNgPnp2ndFwdBwd.monitoring.inHomePos,
                           commands := "Unit1.Em5.HmiInterface".cmCathodeMainPnP1AxisX.commands,
                           interlockOk := "Unit1.Em5.ControlNodes".cm.Interlock.cathodeMainPnP1AxisX.source.posAbsolute,
                           intOut := "Unit1.Em5.HmiInterface".intCondition.Axis_07.Position.intOut);
   #_w1 := (NOT (NOT "Unit1.Em5.ControlNodes".mainPnP."step".action1[1070] AND NOT "Unit1.Em5.ControlNodes".mainPnP."step".action1[112] AND NOT "Unit1.Em5.ControlNodes".mainPnP."step".action1[130] AND NOT "Unit1.Em5.ControlNodes".mainPnP."step".action1[180] AND NOT "Unit1.Em5.ControlNodes".mainPnP."step".action1[420] AND NOT "Unit1.Em5.ControlNodes".mainPnP."step".action1[520]) OR NOT (NOT "Unit1.Em5.ControlNodes".mainPnP."step".action1[220] AND NOT "Unit1.Em5.ControlNodes".mainPnP."step".action1[720]) OR NOT (NOT "Unit1.Em5.ControlNodes".gaugeRnR."step".action1[510])) AND "Unit1.Em5.ControlNodes".cm.Interlock.cathodeMainPnP1AxisX.source.posAbsolute[0];
   IF #_w1 THEN "Unit1.Em5.ControlNodes".cmCathodeMainPnP1AxisX.commands.selectSetPosition := 0; END_IF;
   "Unit1.Em5.ControlNodes".cm.axisCommand.cathodeMainPnP1AxisX.posAbsolute[0] := #_w1;
END_REGION

REGION Network 82: CmCathodeMainPnP1AxisX Position Absolute Position1
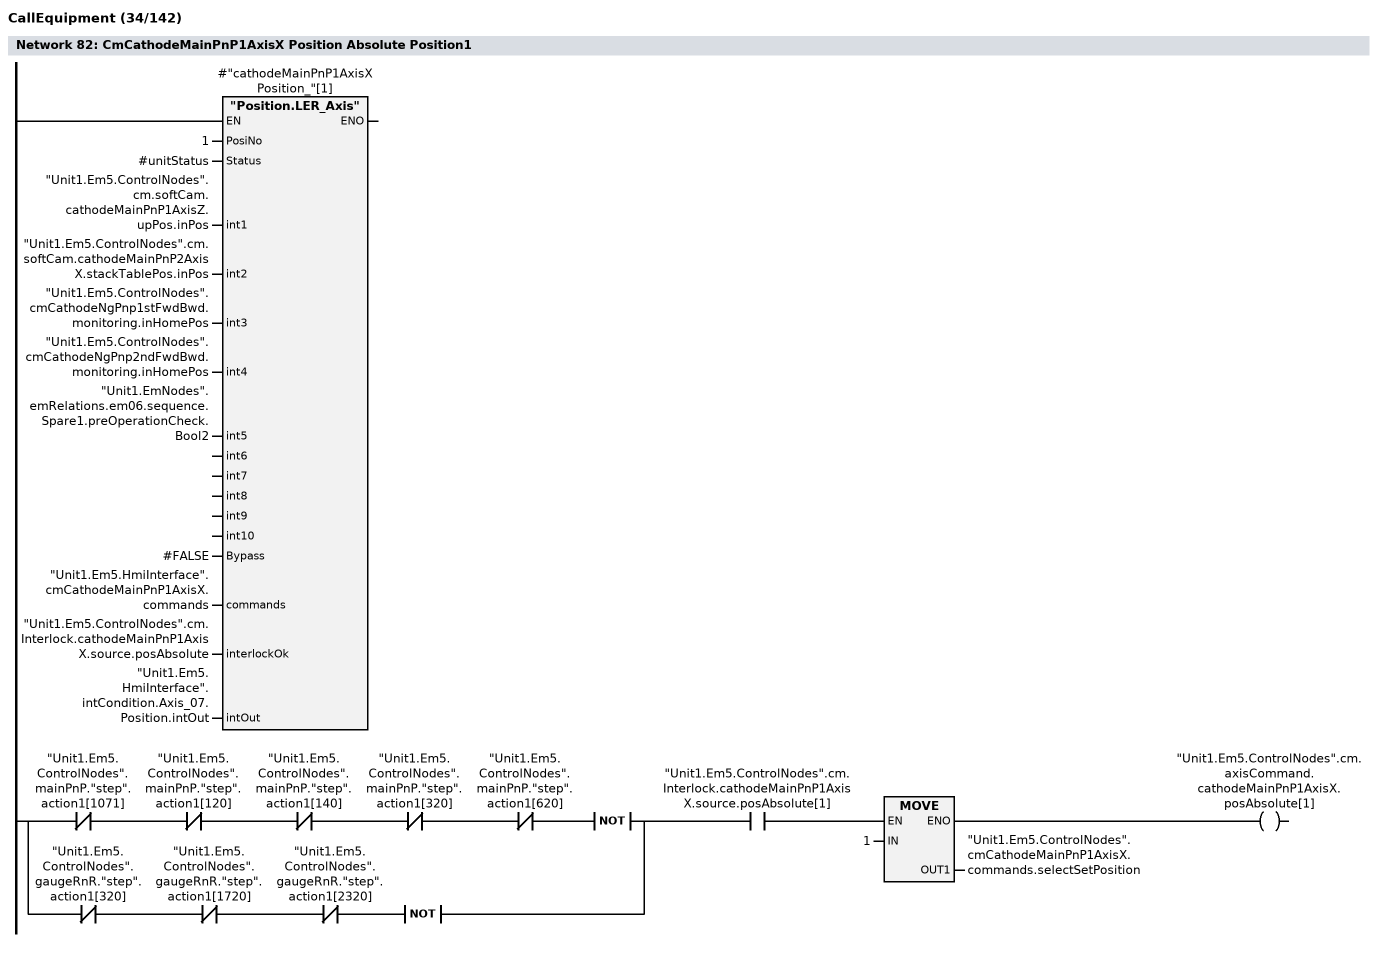
   RUNG wire#powerrail
      #"cathodeMainPnP1AxisX Position_"[1](PosiNo := 1, Status := #unitStatus, int1 := "Unit1.Em5.ControlNodes".cm.softCam.cathodeMainPnP1AxisZ.upPos.inPos, int2 := "Unit1.Em5.ControlNodes".cm.softCam.cathodeMainPnP2AxisX.stackTablePos.inPos, int3 := "Unit1.Em5.ControlNodes".cmCathodeNgPnp1stFwdBwd.monitoring.inHomePos, int4 := "Unit1.Em5.ControlNodes".cmCathodeNgPnp2ndFwdBwd.monitoring.inHomePos, int5 := "Unit1.EmNodes".emRelations.em06.sequence.Spare1.preOperationCheck.Bool2, int6 :=, int7 :=, int8 :=, int9 :=, int10 :=, Bypass := #FALSE, commands := "Unit1.Em5.HmiInterface".cmCathodeMainPnP1AxisX.commands, interlockOk := "Unit1.Em5.ControlNodes".cm.Interlock.cathodeMainPnP1AxisX.source.posAbsolute, intOut := "Unit1.Em5.HmiInterface".intCondition.Axis_07.Position.intOut)
   END_RUNG
   RUNG wire#powerrail
      I_Contact( "Unit1.Em5.ControlNodes".mainPnP."step".action1[1071] )
      I_Contact( "Unit1.Em5.ControlNodes".mainPnP."step".action1[120] )
      I_Contact( "Unit1.Em5.ControlNodes".mainPnP."step".action1[140] )
      I_Contact( "Unit1.Em5.ControlNodes".mainPnP."step".action1[320] )
      I_Contact( "Unit1.Em5.ControlNodes".mainPnP."step".action1[620] )
      Not()
      wire#w1
      Contact( "Unit1.Em5.ControlNodes".cm.Interlock.cathodeMainPnP1AxisX.source.posAbsolute[1] )
      Move(in := 1, out1 => "Unit1.Em5.ControlNodes".cmCathodeMainPnP1AxisX.commands.selectSetPosition)
      Coil( "Unit1.Em5.ControlNodes".cm.axisCommand.cathodeMainPnP1AxisX.posAbsolute[1] )
   END_RUNG
   RUNG wire#powerrail
      I_Contact( "Unit1.Em5.ControlNodes".gaugeRnR."step".action1[320] )
      I_Contact( "Unit1.Em5.ControlNodes".gaugeRnR."step".action1[1720] )
      I_Contact( "Unit1.Em5.ControlNodes".gaugeRnR."step".action1[2320] )
      Not()
   END_RUNG wire#w1
   // the same network as SCL:
   #"cathodeMainPnP1AxisX Position_"[1](PosiNo := 1,   // "Position.LER_Axis"
                           Status := #unitStatus,
                           int1 := "Unit1.Em5.ControlNodes".cm.softCam.cathodeMainPnP1AxisZ.upPos.inPos,
                           int2 := "Unit1.Em5.ControlNodes".cm.softCam.cathodeMainPnP2AxisX.stackTablePos.inPos,
                           int3 := "Unit1.Em5.ControlNodes".cmCathodeNgPnp1stFwdBwd.monitoring.inHomePos,
                           int4 := "Unit1.Em5.ControlNodes".cmCathodeNgPnp2ndFwdBwd.monitoring.inHomePos,
                           int5 := "Unit1.EmNodes".emRelations.em06.sequence.Spare1.preOperationCheck.Bool2,
                           Bypass := #FALSE,
                           commands := "Unit1.Em5.HmiInterface".cmCathodeMainPnP1AxisX.commands,
                           interlockOk := "Unit1.Em5.ControlNodes".cm.Interlock.cathodeMainPnP1AxisX.source.posAbsolute,
                           intOut := "Unit1.Em5.HmiInterface".intCondition.Axis_07.Position.intOut);
   #_w1 := (NOT (NOT "Unit1.Em5.ControlNodes".mainPnP."step".action1[1071] AND NOT "Unit1.Em5.ControlNodes".mainPnP."step".action1[120] AND NOT "Unit1.Em5.ControlNodes".mainPnP."step".action1[140] AND NOT "Unit1.Em5.ControlNodes".mainPnP."step".action1[320] AND NOT "Unit1.Em5.ControlNodes".mainPnP."step".action1[620]) OR NOT (NOT "Unit1.Em5.ControlNodes".gaugeRnR."step".action1[320] AND NOT "Unit1.Em5.ControlNodes".gaugeRnR."step".action1[1720] AND NOT "Unit1.Em5.ControlNodes".gaugeRnR."step".action1[2320])) AND "Unit1.Em5.ControlNodes".cm.Interlock.cathodeMainPnP1AxisX.source.posAbsolute[1];
   IF #_w1 THEN "Unit1.Em5.ControlNodes".cmCathodeMainPnP1AxisX.commands.selectSetPosition := 1; END_IF;
   "Unit1.Em5.ControlNodes".cm.axisCommand.cathodeMainPnP1AxisX.posAbsolute[1] := #_w1;
END_REGION

REGION Network 83: CmCathodeMainPnP1AxisX Position Absolute Position2
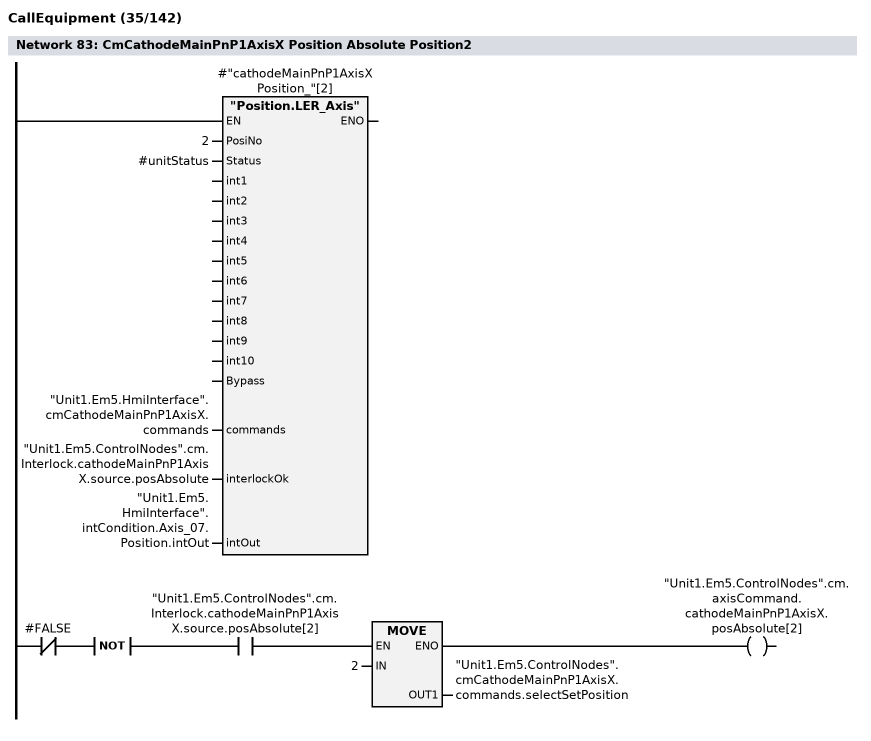
   RUNG wire#powerrail
      #"cathodeMainPnP1AxisX Position_"[2](PosiNo := 2, Status := #unitStatus, int1 :=, int2 :=, int3 :=, int4 :=, int5 :=, int6 :=, int7 :=, int8 :=, int9 :=, int10 :=, Bypass :=, commands := "Unit1.Em5.HmiInterface".cmCathodeMainPnP1AxisX.commands, interlockOk := "Unit1.Em5.ControlNodes".cm.Interlock.cathodeMainPnP1AxisX.source.posAbsolute, intOut := "Unit1.Em5.HmiInterface".intCondition.Axis_07.Position.intOut)
   END_RUNG
   RUNG wire#powerrail
      I_Contact( #FALSE )
      Not()
      Contact( "Unit1.Em5.ControlNodes".cm.Interlock.cathodeMainPnP1AxisX.source.posAbsolute[2] )
      Move(in := 2, out1 => "Unit1.Em5.ControlNodes".cmCathodeMainPnP1AxisX.commands.selectSetPosition)
      Coil( "Unit1.Em5.ControlNodes".cm.axisCommand.cathodeMainPnP1AxisX.posAbsolute[2] )
   END_RUNG
   // the same network as SCL:
   #"cathodeMainPnP1AxisX Position_"[2](PosiNo := 2,   // "Position.LER_Axis"
                           Status := #unitStatus,
                           commands := "Unit1.Em5.HmiInterface".cmCathodeMainPnP1AxisX.commands,
                           interlockOk := "Unit1.Em5.ControlNodes".cm.Interlock.cathodeMainPnP1AxisX.source.posAbsolute,
                           intOut := "Unit1.Em5.HmiInterface".intCondition.Axis_07.Position.intOut);
   #_w1 := NOT (NOT #FALSE) AND "Unit1.Em5.ControlNodes".cm.Interlock.cathodeMainPnP1AxisX.source.posAbsolute[2];
   IF #_w1 THEN "Unit1.Em5.ControlNodes".cmCathodeMainPnP1AxisX.commands.selectSetPosition := 2; END_IF;
   "Unit1.Em5.ControlNodes".cm.axisCommand.cathodeMainPnP1AxisX.posAbsolute[2] := #_w1;
END_REGION

REGION Network 84: CmCathodeMainPnP1AxisX Position Absolute Position3
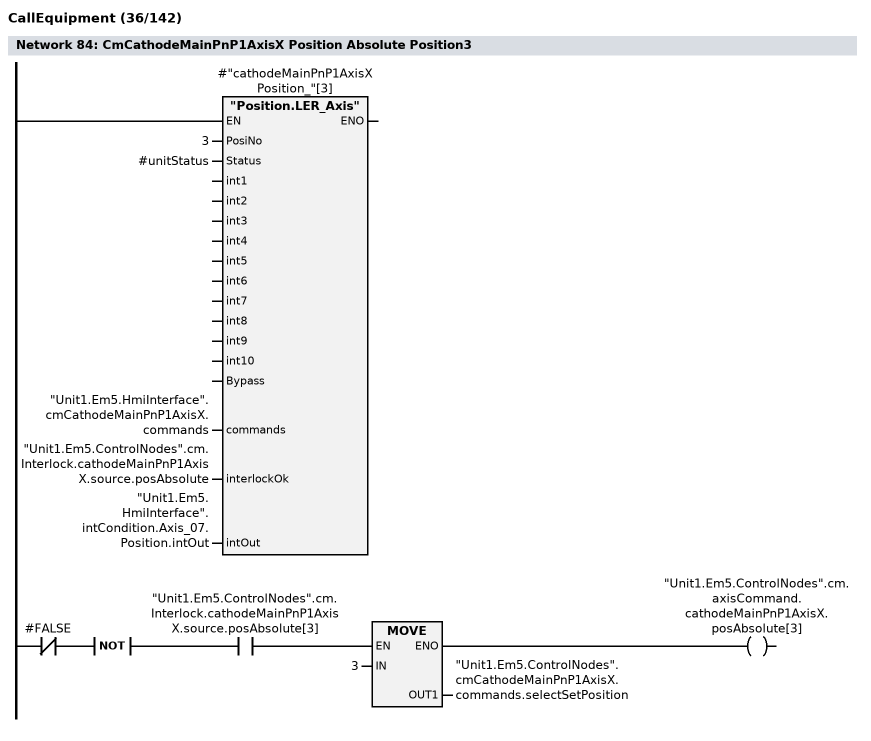
   RUNG wire#powerrail
      #"cathodeMainPnP1AxisX Position_"[3](PosiNo := 3, Status := #unitStatus, int1 :=, int2 :=, int3 :=, int4 :=, int5 :=, int6 :=, int7 :=, int8 :=, int9 :=, int10 :=, Bypass :=, commands := "Unit1.Em5.HmiInterface".cmCathodeMainPnP1AxisX.commands, interlockOk := "Unit1.Em5.ControlNodes".cm.Interlock.cathodeMainPnP1AxisX.source.posAbsolute, intOut := "Unit1.Em5.HmiInterface".intCondition.Axis_07.Position.intOut)
   END_RUNG
   RUNG wire#powerrail
      I_Contact( #FALSE )
      Not()
      Contact( "Unit1.Em5.ControlNodes".cm.Interlock.cathodeMainPnP1AxisX.source.posAbsolute[3] )
      Move(in := 3, out1 => "Unit1.Em5.ControlNodes".cmCathodeMainPnP1AxisX.commands.selectSetPosition)
      Coil( "Unit1.Em5.ControlNodes".cm.axisCommand.cathodeMainPnP1AxisX.posAbsolute[3] )
   END_RUNG
   // the same network as SCL:
   #"cathodeMainPnP1AxisX Position_"[3](PosiNo := 3,   // "Position.LER_Axis"
                           Status := #unitStatus,
                           commands := "Unit1.Em5.HmiInterface".cmCathodeMainPnP1AxisX.commands,
                           interlockOk := "Unit1.Em5.ControlNodes".cm.Interlock.cathodeMainPnP1AxisX.source.posAbsolute,
                           intOut := "Unit1.Em5.HmiInterface".intCondition.Axis_07.Position.intOut);
   #_w1 := NOT (NOT #FALSE) AND "Unit1.Em5.ControlNodes".cm.Interlock.cathodeMainPnP1AxisX.source.posAbsolute[3];
   IF #_w1 THEN "Unit1.Em5.ControlNodes".cmCathodeMainPnP1AxisX.commands.selectSetPosition := 3; END_IF;
   "Unit1.Em5.ControlNodes".cm.axisCommand.cathodeMainPnP1AxisX.posAbsolute[3] := #_w1;
END_REGION

REGION Network 85: CmCathodeMainPnP1AxisX Position Absolute Position4
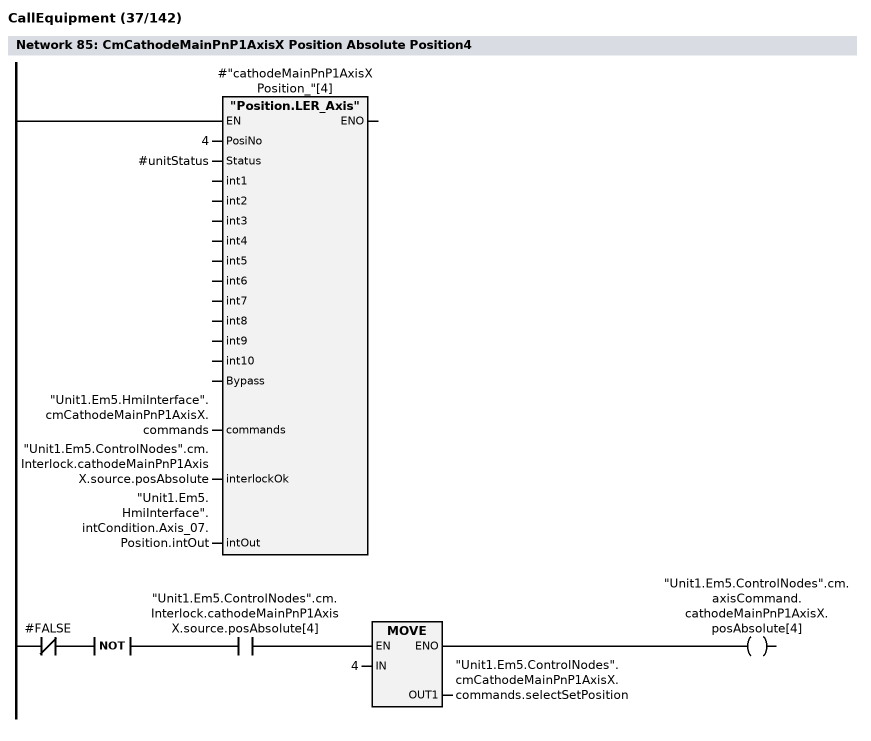
   RUNG wire#powerrail
      #"cathodeMainPnP1AxisX Position_"[4](PosiNo := 4, Status := #unitStatus, int1 :=, int2 :=, int3 :=, int4 :=, int5 :=, int6 :=, int7 :=, int8 :=, int9 :=, int10 :=, Bypass :=, commands := "Unit1.Em5.HmiInterface".cmCathodeMainPnP1AxisX.commands, interlockOk := "Unit1.Em5.ControlNodes".cm.Interlock.cathodeMainPnP1AxisX.source.posAbsolute, intOut := "Unit1.Em5.HmiInterface".intCondition.Axis_07.Position.intOut)
   END_RUNG
   RUNG wire#powerrail
      I_Contact( #FALSE )
      Not()
      Contact( "Unit1.Em5.ControlNodes".cm.Interlock.cathodeMainPnP1AxisX.source.posAbsolute[4] )
      Move(in := 4, out1 => "Unit1.Em5.ControlNodes".cmCathodeMainPnP1AxisX.commands.selectSetPosition)
      Coil( "Unit1.Em5.ControlNodes".cm.axisCommand.cathodeMainPnP1AxisX.posAbsolute[4] )
   END_RUNG
   // the same network as SCL:
   #"cathodeMainPnP1AxisX Position_"[4](PosiNo := 4,   // "Position.LER_Axis"
                           Status := #unitStatus,
                           commands := "Unit1.Em5.HmiInterface".cmCathodeMainPnP1AxisX.commands,
                           interlockOk := "Unit1.Em5.ControlNodes".cm.Interlock.cathodeMainPnP1AxisX.source.posAbsolute,
                           intOut := "Unit1.Em5.HmiInterface".intCondition.Axis_07.Position.intOut);
   #_w1 := NOT (NOT #FALSE) AND "Unit1.Em5.ControlNodes".cm.Interlock.cathodeMainPnP1AxisX.source.posAbsolute[4];
   IF #_w1 THEN "Unit1.Em5.ControlNodes".cmCathodeMainPnP1AxisX.commands.selectSetPosition := 4; END_IF;
   "Unit1.Em5.ControlNodes".cm.axisCommand.cathodeMainPnP1AxisX.posAbsolute[4] := #_w1;
END_REGION

REGION Network 86: CmCathodeMainPnP1AxisX Position Absolute Position5
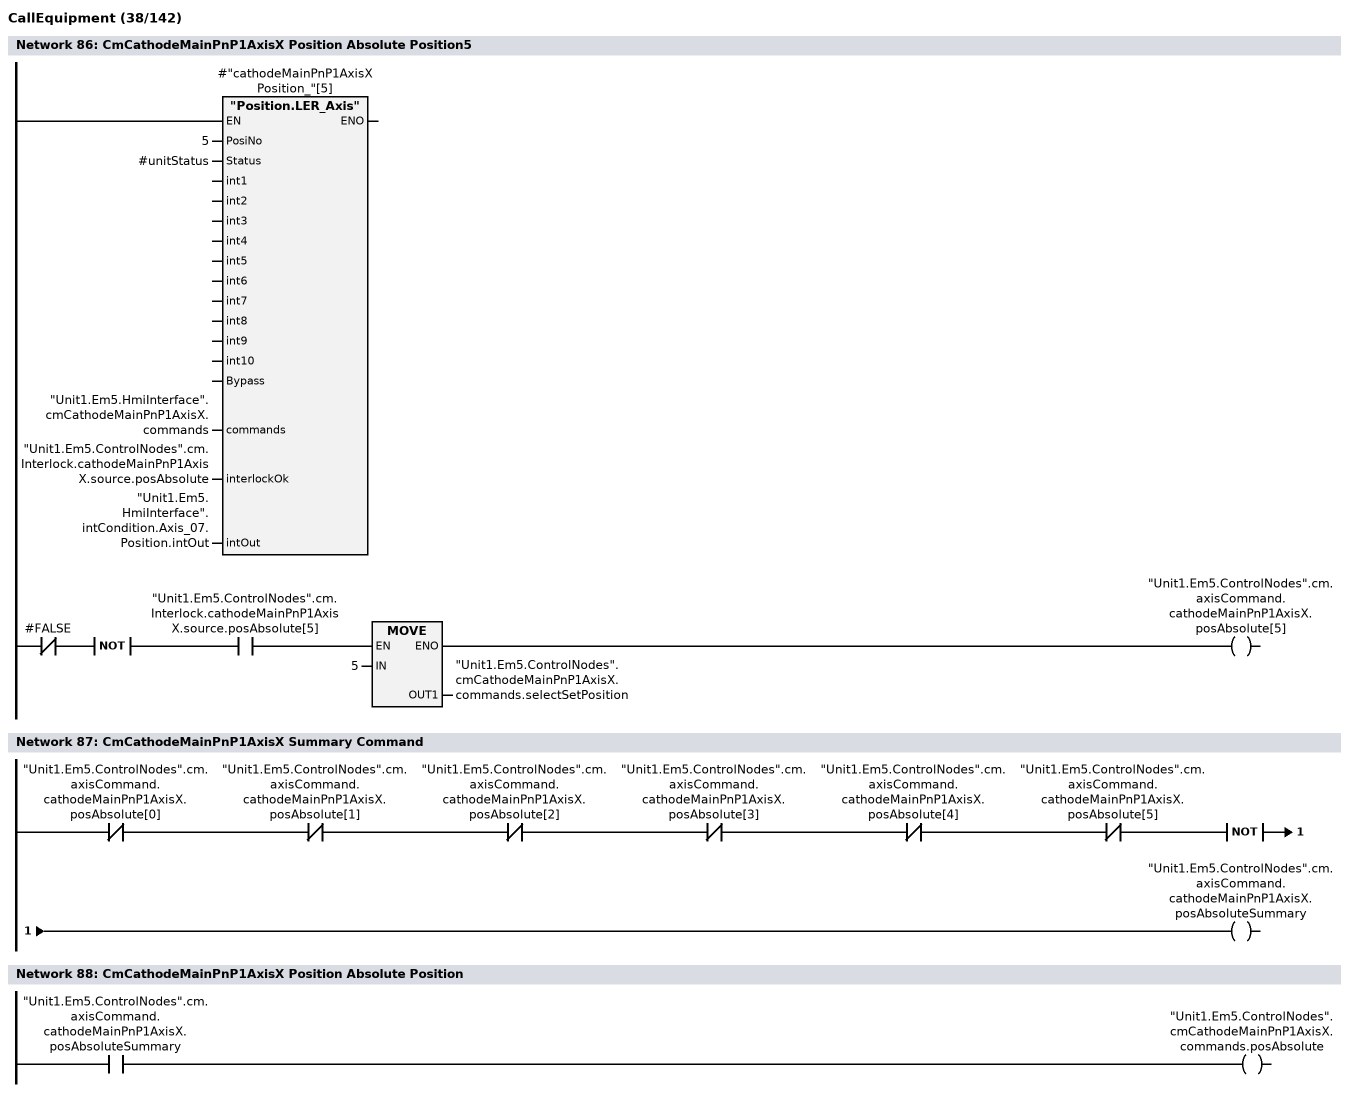
   RUNG wire#powerrail
      #"cathodeMainPnP1AxisX Position_"[5](PosiNo := 5, Status := #unitStatus, int1 :=, int2 :=, int3 :=, int4 :=, int5 :=, int6 :=, int7 :=, int8 :=, int9 :=, int10 :=, Bypass :=, commands := "Unit1.Em5.HmiInterface".cmCathodeMainPnP1AxisX.commands, interlockOk := "Unit1.Em5.ControlNodes".cm.Interlock.cathodeMainPnP1AxisX.source.posAbsolute, intOut := "Unit1.Em5.HmiInterface".intCondition.Axis_07.Position.intOut)
   END_RUNG
   RUNG wire#powerrail
      I_Contact( #FALSE )
      Not()
      Contact( "Unit1.Em5.ControlNodes".cm.Interlock.cathodeMainPnP1AxisX.source.posAbsolute[5] )
      Move(in := 5, out1 => "Unit1.Em5.ControlNodes".cmCathodeMainPnP1AxisX.commands.selectSetPosition)
      Coil( "Unit1.Em5.ControlNodes".cm.axisCommand.cathodeMainPnP1AxisX.posAbsolute[5] )
   END_RUNG
   // the same network as SCL:
   #"cathodeMainPnP1AxisX Position_"[5](PosiNo := 5,   // "Position.LER_Axis"
                           Status := #unitStatus,
                           commands := "Unit1.Em5.HmiInterface".cmCathodeMainPnP1AxisX.commands,
                           interlockOk := "Unit1.Em5.ControlNodes".cm.Interlock.cathodeMainPnP1AxisX.source.posAbsolute,
                           intOut := "Unit1.Em5.HmiInterface".intCondition.Axis_07.Position.intOut);
   #_w1 := NOT (NOT #FALSE) AND "Unit1.Em5.ControlNodes".cm.Interlock.cathodeMainPnP1AxisX.source.posAbsolute[5];
   IF #_w1 THEN "Unit1.Em5.ControlNodes".cmCathodeMainPnP1AxisX.commands.selectSetPosition := 5; END_IF;
   "Unit1.Em5.ControlNodes".cm.axisCommand.cathodeMainPnP1AxisX.posAbsolute[5] := #_w1;
END_REGION

REGION Network 87: CmCathodeMainPnP1AxisX Summary Command
   RUNG wire#powerrail
      I_Contact( "Unit1.Em5.ControlNodes".cm.axisCommand.cathodeMainPnP1AxisX.posAbsolute[0] )
      I_Contact( "Unit1.Em5.ControlNodes".cm.axisCommand.cathodeMainPnP1AxisX.posAbsolute[1] )
      I_Contact( "Unit1.Em5.ControlNodes".cm.axisCommand.cathodeMainPnP1AxisX.posAbsolute[2] )
      I_Contact( "Unit1.Em5.ControlNodes".cm.axisCommand.cathodeMainPnP1AxisX.posAbsolute[3] )
      I_Contact( "Unit1.Em5.ControlNodes".cm.axisCommand.cathodeMainPnP1AxisX.posAbsolute[4] )
      I_Contact( "Unit1.Em5.ControlNodes".cm.axisCommand.cathodeMainPnP1AxisX.posAbsolute[5] )
      Not()
      Coil( "Unit1.Em5.ControlNodes".cm.axisCommand.cathodeMainPnP1AxisX.posAbsoluteSummary )
   END_RUNG
   // the same network as SCL:
   "Unit1.Em5.ControlNodes".cm.axisCommand.cathodeMainPnP1AxisX.posAbsoluteSummary := NOT (NOT "Unit1.Em5.ControlNodes".cm.axisCommand.cathodeMainPnP1AxisX.posAbsolute[0] AND NOT "Unit1.Em5.ControlNodes".cm.axisCommand.cathodeMainPnP1AxisX.posAbsolute[1] AND NOT "Unit1.Em5.ControlNodes".cm.axisCommand.cathodeMainPnP1AxisX.posAbsolute[2] AND NOT "Unit1.Em5.ControlNodes".cm.axisCommand.cathodeMainPnP1AxisX.posAbsolute[3] AND NOT "Unit1.Em5.ControlNodes".cm.axisCommand.cathodeMainPnP1AxisX.posAbsolute[4] AND NOT "Unit1.Em5.ControlNodes".cm.axisCommand.cathodeMainPnP1AxisX.posAbsolute[5]);
END_REGION

REGION Network 88: CmCathodeMainPnP1AxisX Position Absolute Position
   RUNG wire#powerrail
      Contact( "Unit1.Em5.ControlNodes".cm.axisCommand.cathodeMainPnP1AxisX.posAbsoluteSummary )
      Coil( "Unit1.Em5.ControlNodes".cmCathodeMainPnP1AxisX.commands.posAbsolute )
   END_RUNG
   // the same network as SCL:
   "Unit1.Em5.ControlNodes".cmCathodeMainPnP1AxisX.commands.posAbsolute := "Unit1.Em5.ControlNodes".cm.axisCommand.cathodeMainPnP1AxisX.posAbsoluteSummary;
END_REGION

REGION Network 89: CmCathodeMainPnP1AxisX Interlock Summary
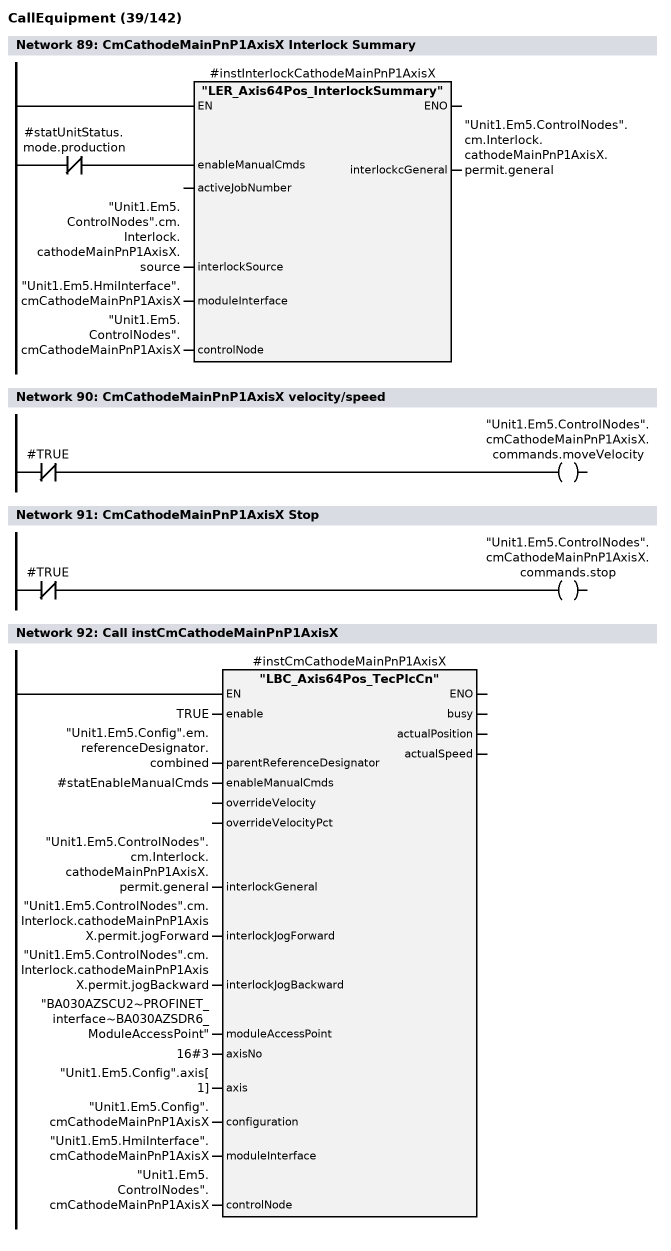
   RUNG wire#powerrail
      #instInterlockCathodeMainPnP1AxisX(enableManualCmds := wire#w1, activeJobNumber :=, interlockSource := "Unit1.Em5.ControlNodes".cm.Interlock.cathodeMainPnP1AxisX.source, moduleInterface := "Unit1.Em5.HmiInterface".cmCathodeMainPnP1AxisX, controlNode := "Unit1.Em5.ControlNodes".cmCathodeMainPnP1AxisX, interlockcGeneral => "Unit1.Em5.ControlNodes".cm.Interlock.cathodeMainPnP1AxisX.permit.general)
   END_RUNG
   RUNG wire#powerrail
      I_Contact( #statUnitStatus.mode.production )
   END_RUNG wire#w1
   // the same network as SCL:
   #instInterlockCathodeMainPnP1AxisX(enableManualCmds := NOT #statUnitStatus.mode.production,   // "LER_Axis64Pos_InterlockSummary"
                           interlockSource := "Unit1.Em5.ControlNodes".cm.Interlock.cathodeMainPnP1AxisX.source,
                           moduleInterface := "Unit1.Em5.HmiInterface".cmCathodeMainPnP1AxisX,
                           controlNode := "Unit1.Em5.ControlNodes".cmCathodeMainPnP1AxisX,
                           interlockcGeneral => "Unit1.Em5.ControlNodes".cm.Interlock.cathodeMainPnP1AxisX.permit.general);
END_REGION

REGION Network 90: CmCathodeMainPnP1AxisX velocity/speed
   RUNG wire#powerrail
      I_Contact( #TRUE )
      Coil( "Unit1.Em5.ControlNodes".cmCathodeMainPnP1AxisX.commands.moveVelocity )
   END_RUNG
   // the same network as SCL:
   "Unit1.Em5.ControlNodes".cmCathodeMainPnP1AxisX.commands.moveVelocity := NOT #TRUE;
END_REGION

REGION Network 91: CmCathodeMainPnP1AxisX Stop
   RUNG wire#powerrail
      I_Contact( #TRUE )
      Coil( "Unit1.Em5.ControlNodes".cmCathodeMainPnP1AxisX.commands.stop )
   END_RUNG
   // the same network as SCL:
   "Unit1.Em5.ControlNodes".cmCathodeMainPnP1AxisX.commands.stop := NOT #TRUE;
END_REGION

REGION Network 92: Call instCmCathodeMainPnP1AxisX
   RUNG wire#powerrail
      #instCmCathodeMainPnP1AxisX(enable := TRUE, parentReferenceDesignator := "Unit1.Em5.Config".em.referenceDesignator.combined, enableManualCmds := #statEnableManualCmds, overrideVelocity :=, overrideVelocityPct :=, interlockGeneral := "Unit1.Em5.ControlNodes".cm.Interlock.cathodeMainPnP1AxisX.permit.general, interlockJogForward := "Unit1.Em5.ControlNodes".cm.Interlock.cathodeMainPnP1AxisX.permit.jogForward, interlockJogBackward := "Unit1.Em5.ControlNodes".cm.Interlock.cathodeMainPnP1AxisX.permit.jogBackward, moduleAccessPoint := "BA030AZSCU2~PROFINET_interface~BA030AZSDR6_ModuleAccessPoint", axisNo := 16#3, axis := "Unit1.Em5.Config".axis[1], configuration := "Unit1.Em5.Config".cmCathodeMainPnP1AxisX, moduleInterface := "Unit1.Em5.HmiInterface".cmCathodeMainPnP1AxisX, controlNode := "Unit1.Em5.ControlNodes".cmCathodeMainPnP1AxisX, busy =>, actualPosition =>, actualSpeed =>)
   END_RUNG
   // the same network as SCL:
   #instCmCathodeMainPnP1AxisX(enable := TRUE,   // "LBC_Axis64Pos_TecPlcCn"
                           parentReferenceDesignator := "Unit1.Em5.Config".em.referenceDesignator.combined,
                           enableManualCmds := #statEnableManualCmds,
                           interlockGeneral := "Unit1.Em5.ControlNodes".cm.Interlock.cathodeMainPnP1AxisX.permit.general,
                           interlockJogForward := "Unit1.Em5.ControlNodes".cm.Interlock.cathodeMainPnP1AxisX.permit.jogForward,
                           interlockJogBackward := "Unit1.Em5.ControlNodes".cm.Interlock.cathodeMainPnP1AxisX.permit.jogBackward,
                           moduleAccessPoint := "BA030AZSCU2~PROFINET_interface~BA030AZSDR6_ModuleAccessPoint",
                           axisNo := 16#3,
                           axis := "Unit1.Em5.Config".axis[1],
                           configuration := "Unit1.Em5.Config".cmCathodeMainPnP1AxisX,
                           moduleInterface := "Unit1.Em5.HmiInterface".cmCathodeMainPnP1AxisX,
                           controlNode := "Unit1.Em5.ControlNodes".cmCathodeMainPnP1AxisX);
END_REGION

REGION Network 93: CmCathodeMainPnP1AxisX SoftCam
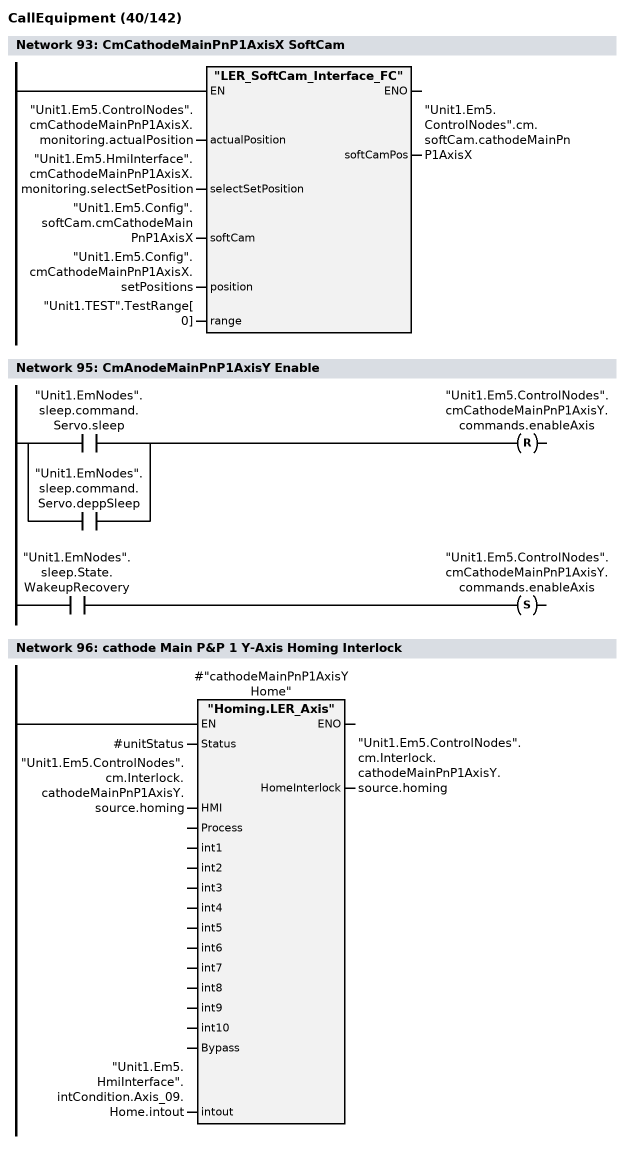
   RUNG wire#powerrail
      "LER_SoftCam_Interface_FC"(actualPosition := "Unit1.Em5.ControlNodes".cmCathodeMainPnP1AxisX.monitoring.actualPosition, selectSetPosition := "Unit1.Em5.HmiInterface".cmCathodeMainPnP1AxisX.monitoring.selectSetPosition, softCam := "Unit1.Em5.Config".softCam.cmCathodeMainPnP1AxisX, position := "Unit1.Em5.Config".cmCathodeMainPnP1AxisX.setPositions, range := "Unit1.TEST".TestRange[0], softCamPos => "Unit1.Em5.ControlNodes".cm.softCam.cathodeMainPnP1AxisX)
   END_RUNG
   // the same network as SCL:
   "LER_SoftCam_Interface_FC"(actualPosition := "Unit1.Em5.ControlNodes".cmCathodeMainPnP1AxisX.monitoring.actualPosition,
                           selectSetPosition := "Unit1.Em5.HmiInterface".cmCathodeMainPnP1AxisX.monitoring.selectSetPosition,
                           softCam := "Unit1.Em5.Config".softCam.cmCathodeMainPnP1AxisX,
                           position := "Unit1.Em5.Config".cmCathodeMainPnP1AxisX.setPositions,
                           range := "Unit1.TEST".TestRange[0],
                           softCamPos => "Unit1.Em5.ControlNodes".cm.softCam.cathodeMainPnP1AxisX);
END_REGION

REGION Network 95: CmAnodeMainPnP1AxisY Enable
   RUNG wire#powerrail
      Contact( "Unit1.EmNodes".sleep.command.Servo.sleep )
      wire#w1
      R_Coil( "Unit1.Em5.ControlNodes".cmCathodeMainPnP1AxisY.commands.enableAxis )
   END_RUNG
   RUNG wire#powerrail
      Contact( "Unit1.EmNodes".sleep.command.Servo.deppSleep )
   END_RUNG wire#w1
   RUNG wire#powerrail
      Contact( "Unit1.EmNodes".sleep.State.WakeupRecovery )
      S_Coil( "Unit1.Em5.ControlNodes".cmCathodeMainPnP1AxisY.commands.enableAxis )
   END_RUNG
   // the same network as SCL:
   IF "Unit1.EmNodes".sleep.command.Servo.sleep OR "Unit1.EmNodes".sleep.command.Servo.deppSleep THEN
       "Unit1.Em5.ControlNodes".cmCathodeMainPnP1AxisY.commands.enableAxis := FALSE;
   END_IF;
   IF "Unit1.EmNodes".sleep.State.WakeupRecovery THEN
       "Unit1.Em5.ControlNodes".cmCathodeMainPnP1AxisY.commands.enableAxis := TRUE;
   END_IF;
END_REGION

REGION Network 96: cathode Main P&P 1 Y-Axis Homing Interlock
   RUNG wire#powerrail
      #"cathodeMainPnP1AxisY Home"(Status := #unitStatus, HMI := "Unit1.Em5.ControlNodes".cm.Interlock.cathodeMainPnP1AxisY.source.homing, Process :=, int1 :=, int2 :=, int3 :=, int4 :=, int5 :=, int6 :=, int7 :=, int8 :=, int9 :=, int10 :=, Bypass :=, intout := "Unit1.Em5.HmiInterface".intCondition.Axis_09.Home.intout, HomeInterlock => "Unit1.Em5.ControlNodes".cm.Interlock.cathodeMainPnP1AxisY.source.homing)
   END_RUNG
   // the same network as SCL:
   #"cathodeMainPnP1AxisY Home"(Status := #unitStatus,   // "Homing.LER_Axis"
                           HMI := "Unit1.Em5.ControlNodes".cm.Interlock.cathodeMainPnP1AxisY.source.homing,
                           intout := "Unit1.Em5.HmiInterface".intCondition.Axis_09.Home.intout,
                           HomeInterlock => "Unit1.Em5.ControlNodes".cm.Interlock.cathodeMainPnP1AxisY.source.homing);
END_REGION

REGION Network 97: CmCathodeMainPnP1AxisY Position Absolute Jog
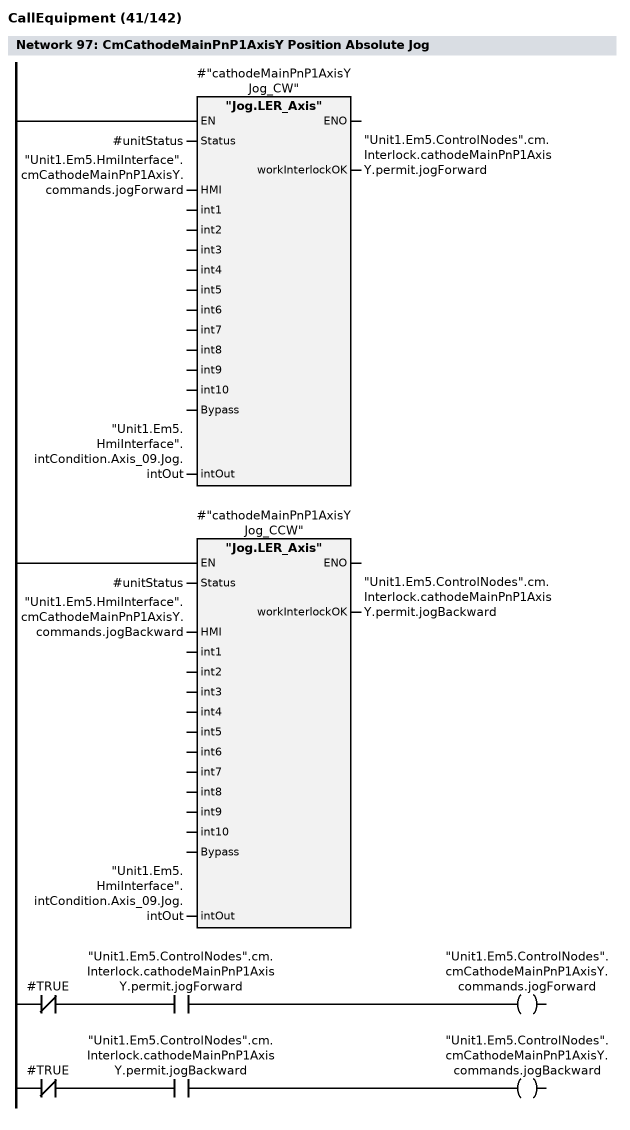
   RUNG wire#powerrail
      #"cathodeMainPnP1AxisY Jog_CW"(Status := #unitStatus, HMI := "Unit1.Em5.HmiInterface".cmCathodeMainPnP1AxisY.commands.jogForward, int1 :=, int2 :=, int3 :=, int4 :=, int5 :=, int6 :=, int7 :=, int8 :=, int9 :=, int10 :=, Bypass :=, intOut := "Unit1.Em5.HmiInterface".intCondition.Axis_09.Jog.intOut, workInterlockOK => "Unit1.Em5.ControlNodes".cm.Interlock.cathodeMainPnP1AxisY.permit.jogForward)
   END_RUNG
   RUNG wire#powerrail
      #"cathodeMainPnP1AxisY Jog_CCW"(Status := #unitStatus, HMI := "Unit1.Em5.HmiInterface".cmCathodeMainPnP1AxisY.commands.jogBackward, int1 :=, int2 :=, int3 :=, int4 :=, int5 :=, int6 :=, int7 :=, int8 :=, int9 :=, int10 :=, Bypass :=, intOut := "Unit1.Em5.HmiInterface".intCondition.Axis_09.Jog.intOut, workInterlockOK => "Unit1.Em5.ControlNodes".cm.Interlock.cathodeMainPnP1AxisY.permit.jogBackward)
   END_RUNG
   RUNG wire#powerrail
      I_Contact( #TRUE )
      Contact( "Unit1.Em5.ControlNodes".cm.Interlock.cathodeMainPnP1AxisY.permit.jogForward )
      Coil( "Unit1.Em5.ControlNodes".cmCathodeMainPnP1AxisY.commands.jogForward )
   END_RUNG
   RUNG wire#powerrail
      I_Contact( #TRUE )
      Contact( "Unit1.Em5.ControlNodes".cm.Interlock.cathodeMainPnP1AxisY.permit.jogBackward )
      Coil( "Unit1.Em5.ControlNodes".cmCathodeMainPnP1AxisY.commands.jogBackward )
   END_RUNG
   // the same network as SCL:
   #"cathodeMainPnP1AxisY Jog_CW"(Status := #unitStatus,   // "Jog.LER_Axis"
                           HMI := "Unit1.Em5.HmiInterface".cmCathodeMainPnP1AxisY.commands.jogForward,
                           intOut := "Unit1.Em5.HmiInterface".intCondition.Axis_09.Jog.intOut,
                           workInterlockOK => "Unit1.Em5.ControlNodes".cm.Interlock.cathodeMainPnP1AxisY.permit.jogForward);
   #"cathodeMainPnP1AxisY Jog_CCW"(Status := #unitStatus,   // "Jog.LER_Axis"
                           HMI := "Unit1.Em5.HmiInterface".cmCathodeMainPnP1AxisY.commands.jogBackward,
                           intOut := "Unit1.Em5.HmiInterface".intCondition.Axis_09.Jog.intOut,
                           workInterlockOK => "Unit1.Em5.ControlNodes".cm.Interlock.cathodeMainPnP1AxisY.permit.jogBackward);
   "Unit1.Em5.ControlNodes".cmCathodeMainPnP1AxisY.commands.jogForward := NOT #TRUE AND "Unit1.Em5.ControlNodes".cm.Interlock.cathodeMainPnP1AxisY.permit.jogForward;
   "Unit1.Em5.ControlNodes".cmCathodeMainPnP1AxisY.commands.jogBackward := NOT #TRUE AND "Unit1.Em5.ControlNodes".cm.Interlock.cathodeMainPnP1AxisY.permit.jogBackward;
END_REGION

REGION Network 98: CmCathodeMainPnP1AxisY Position Absolute Position0
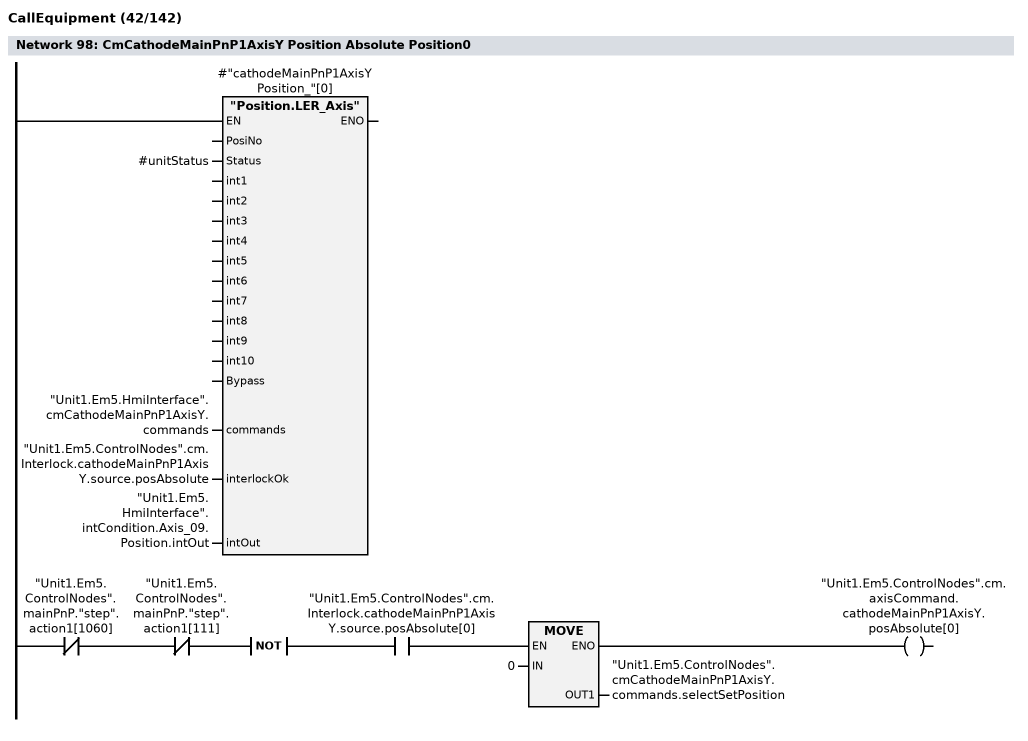
   RUNG wire#powerrail
      #"cathodeMainPnP1AxisY Position_"[0](PosiNo :=, Status := #unitStatus, int1 :=, int2 :=, int3 :=, int4 :=, int5 :=, int6 :=, int7 :=, int8 :=, int9 :=, int10 :=, Bypass :=, commands := "Unit1.Em5.HmiInterface".cmCathodeMainPnP1AxisY.commands, interlockOk := "Unit1.Em5.ControlNodes".cm.Interlock.cathodeMainPnP1AxisY.source.posAbsolute, intOut := "Unit1.Em5.HmiInterface".intCondition.Axis_09.Position.intOut)
   END_RUNG
   RUNG wire#powerrail
      I_Contact( "Unit1.Em5.ControlNodes".mainPnP."step".action1[1060] )
      I_Contact( "Unit1.Em5.ControlNodes".mainPnP."step".action1[111] )
      Not()
      Contact( "Unit1.Em5.ControlNodes".cm.Interlock.cathodeMainPnP1AxisY.source.posAbsolute[0] )
      Move(in := 0, out1 => "Unit1.Em5.ControlNodes".cmCathodeMainPnP1AxisY.commands.selectSetPosition)
      Coil( "Unit1.Em5.ControlNodes".cm.axisCommand.cathodeMainPnP1AxisY.posAbsolute[0] )
   END_RUNG
   // the same network as SCL:
   #"cathodeMainPnP1AxisY Position_"[0](Status := #unitStatus,   // "Position.LER_Axis"
                           commands := "Unit1.Em5.HmiInterface".cmCathodeMainPnP1AxisY.commands,
                           interlockOk := "Unit1.Em5.ControlNodes".cm.Interlock.cathodeMainPnP1AxisY.source.posAbsolute,
                           intOut := "Unit1.Em5.HmiInterface".intCondition.Axis_09.Position.intOut);
   #_w1 := NOT (NOT "Unit1.Em5.ControlNodes".mainPnP."step".action1[1060] AND NOT "Unit1.Em5.ControlNodes".mainPnP."step".action1[111]) AND "Unit1.Em5.ControlNodes".cm.Interlock.cathodeMainPnP1AxisY.source.posAbsolute[0];
   IF #_w1 THEN "Unit1.Em5.ControlNodes".cmCathodeMainPnP1AxisY.commands.selectSetPosition := 0; END_IF;
   "Unit1.Em5.ControlNodes".cm.axisCommand.cathodeMainPnP1AxisY.posAbsolute[0] := #_w1;
END_REGION

REGION Network 99: CmCathodeMainPnP1AxisY Position Absolute Position1
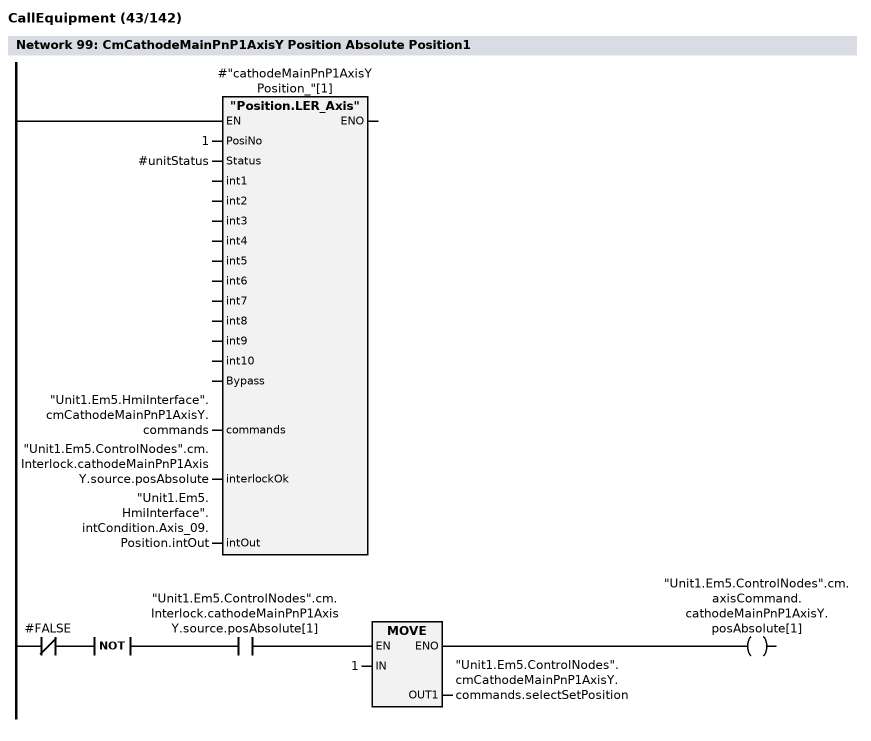
   RUNG wire#powerrail
      #"cathodeMainPnP1AxisY Position_"[1](PosiNo := 1, Status := #unitStatus, int1 :=, int2 :=, int3 :=, int4 :=, int5 :=, int6 :=, int7 :=, int8 :=, int9 :=, int10 :=, Bypass :=, commands := "Unit1.Em5.HmiInterface".cmCathodeMainPnP1AxisY.commands, interlockOk := "Unit1.Em5.ControlNodes".cm.Interlock.cathodeMainPnP1AxisY.source.posAbsolute, intOut := "Unit1.Em5.HmiInterface".intCondition.Axis_09.Position.intOut)
   END_RUNG
   RUNG wire#powerrail
      I_Contact( #FALSE )
      Not()
      Contact( "Unit1.Em5.ControlNodes".cm.Interlock.cathodeMainPnP1AxisY.source.posAbsolute[1] )
      Move(in := 1, out1 => "Unit1.Em5.ControlNodes".cmCathodeMainPnP1AxisY.commands.selectSetPosition)
      Coil( "Unit1.Em5.ControlNodes".cm.axisCommand.cathodeMainPnP1AxisY.posAbsolute[1] )
   END_RUNG
   // the same network as SCL:
   #"cathodeMainPnP1AxisY Position_"[1](PosiNo := 1,   // "Position.LER_Axis"
                           Status := #unitStatus,
                           commands := "Unit1.Em5.HmiInterface".cmCathodeMainPnP1AxisY.commands,
                           interlockOk := "Unit1.Em5.ControlNodes".cm.Interlock.cathodeMainPnP1AxisY.source.posAbsolute,
                           intOut := "Unit1.Em5.HmiInterface".intCondition.Axis_09.Position.intOut);
   #_w1 := NOT (NOT #FALSE) AND "Unit1.Em5.ControlNodes".cm.Interlock.cathodeMainPnP1AxisY.source.posAbsolute[1];
   IF #_w1 THEN "Unit1.Em5.ControlNodes".cmCathodeMainPnP1AxisY.commands.selectSetPosition := 1; END_IF;
   "Unit1.Em5.ControlNodes".cm.axisCommand.cathodeMainPnP1AxisY.posAbsolute[1] := #_w1;
END_REGION

REGION Network 100: CmCathodeMainPnP1AxisY Position Absolute Position2
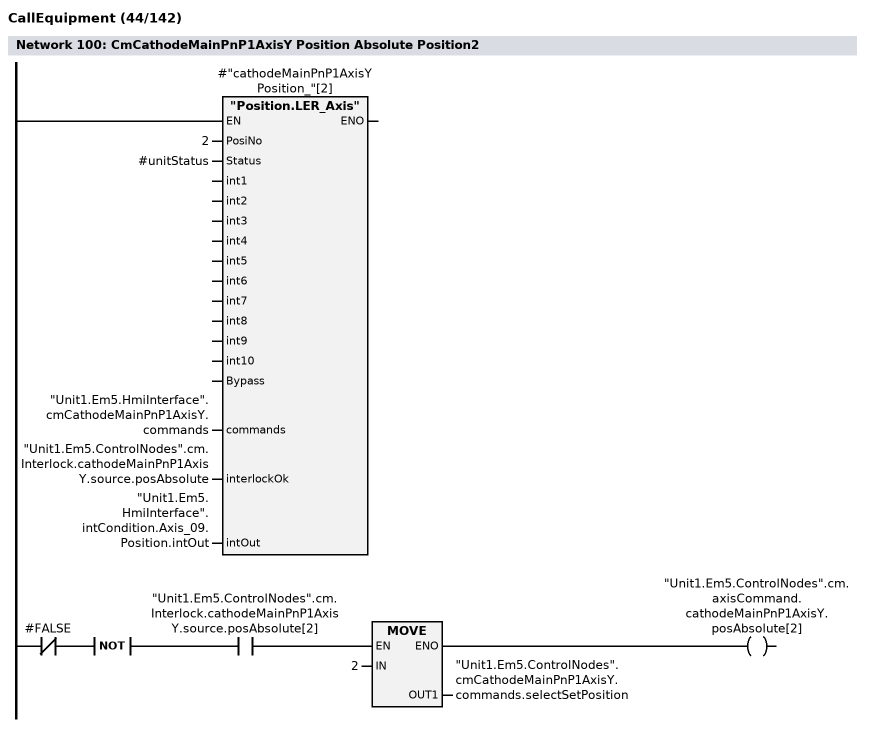
   RUNG wire#powerrail
      #"cathodeMainPnP1AxisY Position_"[2](PosiNo := 2, Status := #unitStatus, int1 :=, int2 :=, int3 :=, int4 :=, int5 :=, int6 :=, int7 :=, int8 :=, int9 :=, int10 :=, Bypass :=, commands := "Unit1.Em5.HmiInterface".cmCathodeMainPnP1AxisY.commands, interlockOk := "Unit1.Em5.ControlNodes".cm.Interlock.cathodeMainPnP1AxisY.source.posAbsolute, intOut := "Unit1.Em5.HmiInterface".intCondition.Axis_09.Position.intOut)
   END_RUNG
   RUNG wire#powerrail
      I_Contact( #FALSE )
      Not()
      Contact( "Unit1.Em5.ControlNodes".cm.Interlock.cathodeMainPnP1AxisY.source.posAbsolute[2] )
      Move(in := 2, out1 => "Unit1.Em5.ControlNodes".cmCathodeMainPnP1AxisY.commands.selectSetPosition)
      Coil( "Unit1.Em5.ControlNodes".cm.axisCommand.cathodeMainPnP1AxisY.posAbsolute[2] )
   END_RUNG
   // the same network as SCL:
   #"cathodeMainPnP1AxisY Position_"[2](PosiNo := 2,   // "Position.LER_Axis"
                           Status := #unitStatus,
                           commands := "Unit1.Em5.HmiInterface".cmCathodeMainPnP1AxisY.commands,
                           interlockOk := "Unit1.Em5.ControlNodes".cm.Interlock.cathodeMainPnP1AxisY.source.posAbsolute,
                           intOut := "Unit1.Em5.HmiInterface".intCondition.Axis_09.Position.intOut);
   #_w1 := NOT (NOT #FALSE) AND "Unit1.Em5.ControlNodes".cm.Interlock.cathodeMainPnP1AxisY.source.posAbsolute[2];
   IF #_w1 THEN "Unit1.Em5.ControlNodes".cmCathodeMainPnP1AxisY.commands.selectSetPosition := 2; END_IF;
   "Unit1.Em5.ControlNodes".cm.axisCommand.cathodeMainPnP1AxisY.posAbsolute[2] := #_w1;
END_REGION

REGION Network 101: CmCathodeMainPnP1AxisY Position Absolute Position3
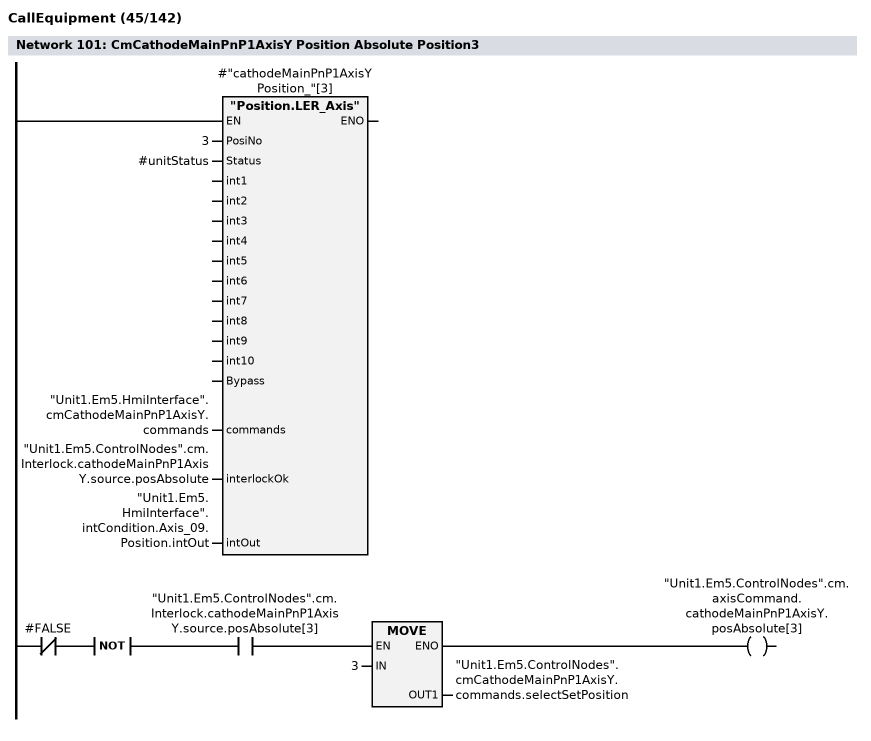
   RUNG wire#powerrail
      #"cathodeMainPnP1AxisY Position_"[3](PosiNo := 3, Status := #unitStatus, int1 :=, int2 :=, int3 :=, int4 :=, int5 :=, int6 :=, int7 :=, int8 :=, int9 :=, int10 :=, Bypass :=, commands := "Unit1.Em5.HmiInterface".cmCathodeMainPnP1AxisY.commands, interlockOk := "Unit1.Em5.ControlNodes".cm.Interlock.cathodeMainPnP1AxisY.source.posAbsolute, intOut := "Unit1.Em5.HmiInterface".intCondition.Axis_09.Position.intOut)
   END_RUNG
   RUNG wire#powerrail
      I_Contact( #FALSE )
      Not()
      Contact( "Unit1.Em5.ControlNodes".cm.Interlock.cathodeMainPnP1AxisY.source.posAbsolute[3] )
      Move(in := 3, out1 => "Unit1.Em5.ControlNodes".cmCathodeMainPnP1AxisY.commands.selectSetPosition)
      Coil( "Unit1.Em5.ControlNodes".cm.axisCommand.cathodeMainPnP1AxisY.posAbsolute[3] )
   END_RUNG
   // the same network as SCL:
   #"cathodeMainPnP1AxisY Position_"[3](PosiNo := 3,   // "Position.LER_Axis"
                           Status := #unitStatus,
                           commands := "Unit1.Em5.HmiInterface".cmCathodeMainPnP1AxisY.commands,
                           interlockOk := "Unit1.Em5.ControlNodes".cm.Interlock.cathodeMainPnP1AxisY.source.posAbsolute,
                           intOut := "Unit1.Em5.HmiInterface".intCondition.Axis_09.Position.intOut);
   #_w1 := NOT (NOT #FALSE) AND "Unit1.Em5.ControlNodes".cm.Interlock.cathodeMainPnP1AxisY.source.posAbsolute[3];
   IF #_w1 THEN "Unit1.Em5.ControlNodes".cmCathodeMainPnP1AxisY.commands.selectSetPosition := 3; END_IF;
   "Unit1.Em5.ControlNodes".cm.axisCommand.cathodeMainPnP1AxisY.posAbsolute[3] := #_w1;
END_REGION

REGION Network 102: CmCathodeMainPnP1AxisY Position Absolute Position4
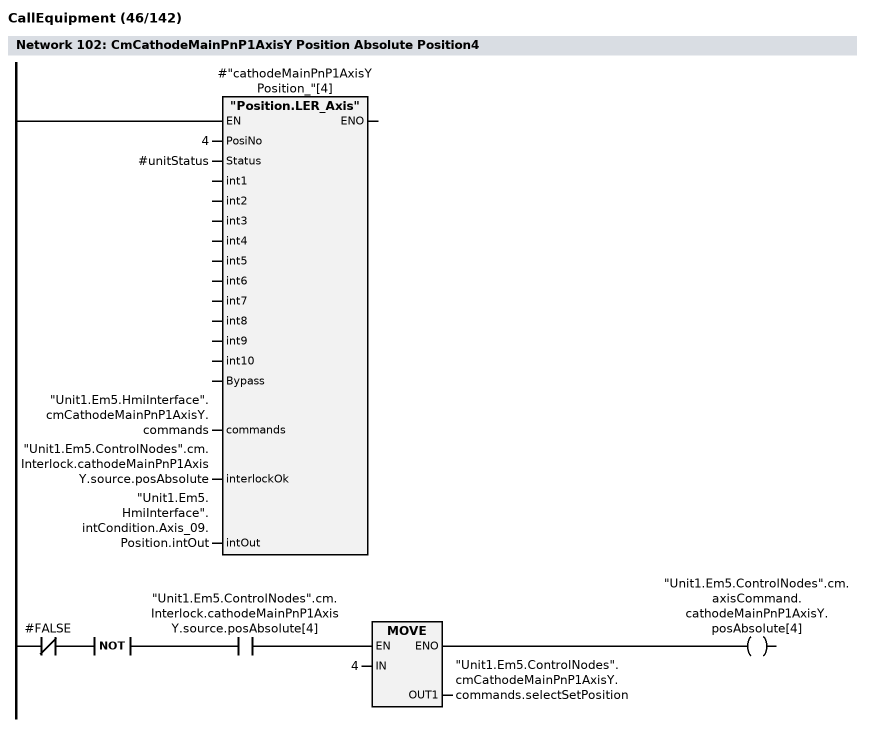
   RUNG wire#powerrail
      #"cathodeMainPnP1AxisY Position_"[4](PosiNo := 4, Status := #unitStatus, int1 :=, int2 :=, int3 :=, int4 :=, int5 :=, int6 :=, int7 :=, int8 :=, int9 :=, int10 :=, Bypass :=, commands := "Unit1.Em5.HmiInterface".cmCathodeMainPnP1AxisY.commands, interlockOk := "Unit1.Em5.ControlNodes".cm.Interlock.cathodeMainPnP1AxisY.source.posAbsolute, intOut := "Unit1.Em5.HmiInterface".intCondition.Axis_09.Position.intOut)
   END_RUNG
   RUNG wire#powerrail
      I_Contact( #FALSE )
      Not()
      Contact( "Unit1.Em5.ControlNodes".cm.Interlock.cathodeMainPnP1AxisY.source.posAbsolute[4] )
      Move(in := 4, out1 => "Unit1.Em5.ControlNodes".cmCathodeMainPnP1AxisY.commands.selectSetPosition)
      Coil( "Unit1.Em5.ControlNodes".cm.axisCommand.cathodeMainPnP1AxisY.posAbsolute[4] )
   END_RUNG
   // the same network as SCL:
   #"cathodeMainPnP1AxisY Position_"[4](PosiNo := 4,   // "Position.LER_Axis"
                           Status := #unitStatus,
                           commands := "Unit1.Em5.HmiInterface".cmCathodeMainPnP1AxisY.commands,
                           interlockOk := "Unit1.Em5.ControlNodes".cm.Interlock.cathodeMainPnP1AxisY.source.posAbsolute,
                           intOut := "Unit1.Em5.HmiInterface".intCondition.Axis_09.Position.intOut);
   #_w1 := NOT (NOT #FALSE) AND "Unit1.Em5.ControlNodes".cm.Interlock.cathodeMainPnP1AxisY.source.posAbsolute[4];
   IF #_w1 THEN "Unit1.Em5.ControlNodes".cmCathodeMainPnP1AxisY.commands.selectSetPosition := 4; END_IF;
   "Unit1.Em5.ControlNodes".cm.axisCommand.cathodeMainPnP1AxisY.posAbsolute[4] := #_w1;
END_REGION

REGION Network 103: CmCathodeMainPnP1AxisY Position Absolute Position5
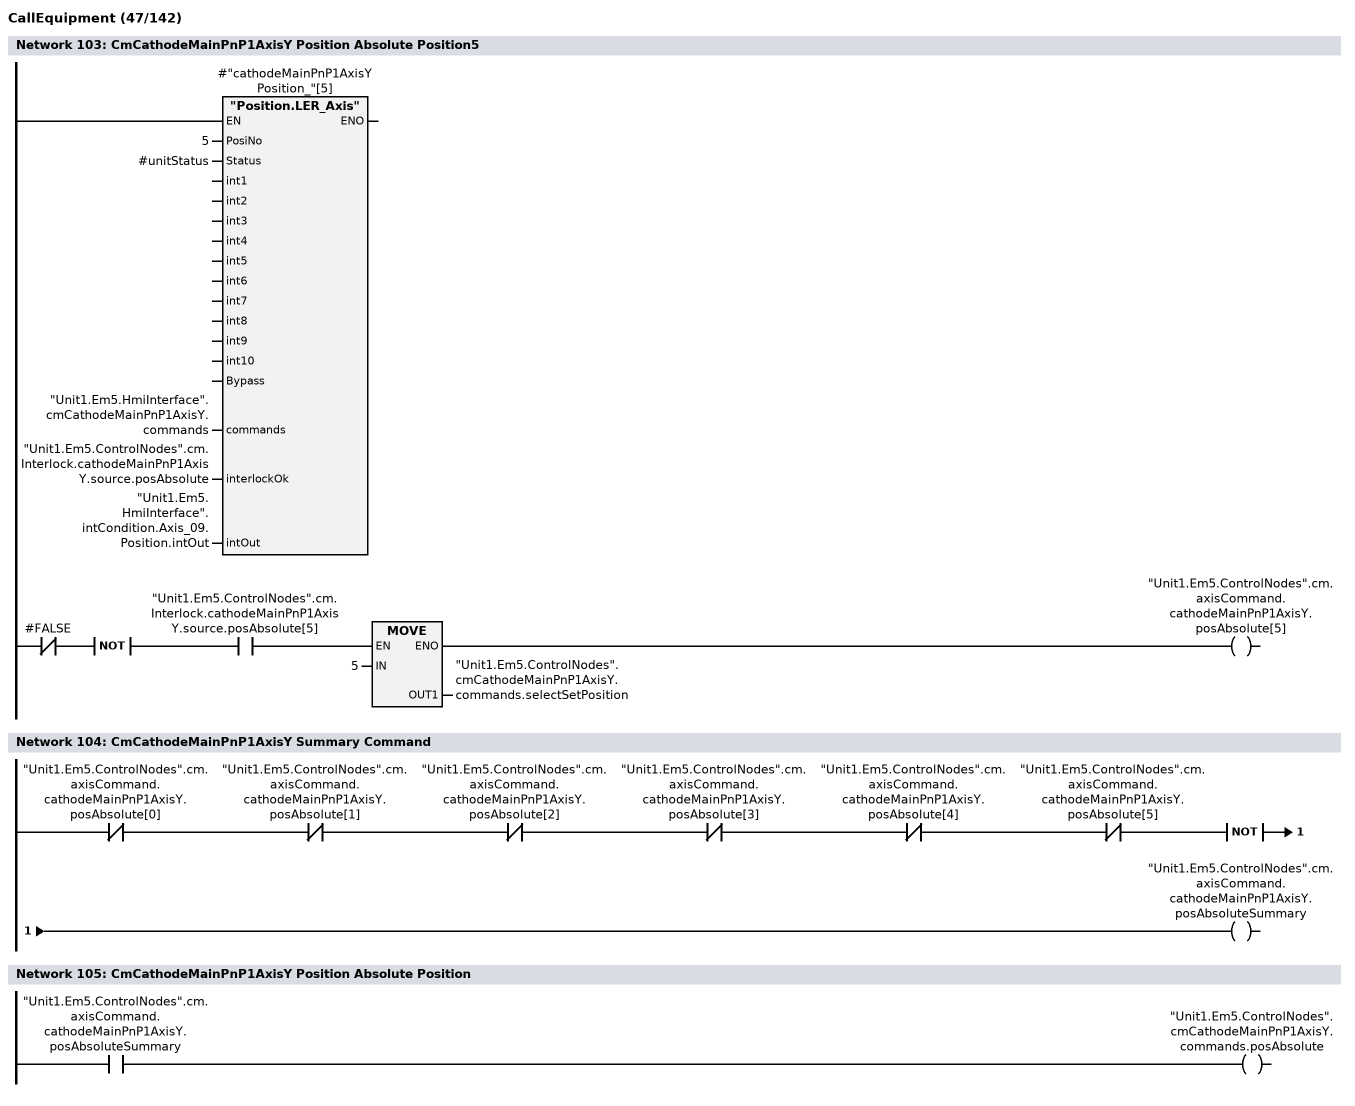
   RUNG wire#powerrail
      #"cathodeMainPnP1AxisY Position_"[5](PosiNo := 5, Status := #unitStatus, int1 :=, int2 :=, int3 :=, int4 :=, int5 :=, int6 :=, int7 :=, int8 :=, int9 :=, int10 :=, Bypass :=, commands := "Unit1.Em5.HmiInterface".cmCathodeMainPnP1AxisY.commands, interlockOk := "Unit1.Em5.ControlNodes".cm.Interlock.cathodeMainPnP1AxisY.source.posAbsolute, intOut := "Unit1.Em5.HmiInterface".intCondition.Axis_09.Position.intOut)
   END_RUNG
   RUNG wire#powerrail
      I_Contact( #FALSE )
      Not()
      Contact( "Unit1.Em5.ControlNodes".cm.Interlock.cathodeMainPnP1AxisY.source.posAbsolute[5] )
      Move(in := 5, out1 => "Unit1.Em5.ControlNodes".cmCathodeMainPnP1AxisY.commands.selectSetPosition)
      Coil( "Unit1.Em5.ControlNodes".cm.axisCommand.cathodeMainPnP1AxisY.posAbsolute[5] )
   END_RUNG
   // the same network as SCL:
   #"cathodeMainPnP1AxisY Position_"[5](PosiNo := 5,   // "Position.LER_Axis"
                           Status := #unitStatus,
                           commands := "Unit1.Em5.HmiInterface".cmCathodeMainPnP1AxisY.commands,
                           interlockOk := "Unit1.Em5.ControlNodes".cm.Interlock.cathodeMainPnP1AxisY.source.posAbsolute,
                           intOut := "Unit1.Em5.HmiInterface".intCondition.Axis_09.Position.intOut);
   #_w1 := NOT (NOT #FALSE) AND "Unit1.Em5.ControlNodes".cm.Interlock.cathodeMainPnP1AxisY.source.posAbsolute[5];
   IF #_w1 THEN "Unit1.Em5.ControlNodes".cmCathodeMainPnP1AxisY.commands.selectSetPosition := 5; END_IF;
   "Unit1.Em5.ControlNodes".cm.axisCommand.cathodeMainPnP1AxisY.posAbsolute[5] := #_w1;
END_REGION

REGION Network 104: CmCathodeMainPnP1AxisY Summary Command
   RUNG wire#powerrail
      I_Contact( "Unit1.Em5.ControlNodes".cm.axisCommand.cathodeMainPnP1AxisY.posAbsolute[0] )
      I_Contact( "Unit1.Em5.ControlNodes".cm.axisCommand.cathodeMainPnP1AxisY.posAbsolute[1] )
      I_Contact( "Unit1.Em5.ControlNodes".cm.axisCommand.cathodeMainPnP1AxisY.posAbsolute[2] )
      I_Contact( "Unit1.Em5.ControlNodes".cm.axisCommand.cathodeMainPnP1AxisY.posAbsolute[3] )
      I_Contact( "Unit1.Em5.ControlNodes".cm.axisCommand.cathodeMainPnP1AxisY.posAbsolute[4] )
      I_Contact( "Unit1.Em5.ControlNodes".cm.axisCommand.cathodeMainPnP1AxisY.posAbsolute[5] )
      Not()
      Coil( "Unit1.Em5.ControlNodes".cm.axisCommand.cathodeMainPnP1AxisY.posAbsoluteSummary )
   END_RUNG
   // the same network as SCL:
   "Unit1.Em5.ControlNodes".cm.axisCommand.cathodeMainPnP1AxisY.posAbsoluteSummary := NOT (NOT "Unit1.Em5.ControlNodes".cm.axisCommand.cathodeMainPnP1AxisY.posAbsolute[0] AND NOT "Unit1.Em5.ControlNodes".cm.axisCommand.cathodeMainPnP1AxisY.posAbsolute[1] AND NOT "Unit1.Em5.ControlNodes".cm.axisCommand.cathodeMainPnP1AxisY.posAbsolute[2] AND NOT "Unit1.Em5.ControlNodes".cm.axisCommand.cathodeMainPnP1AxisY.posAbsolute[3] AND NOT "Unit1.Em5.ControlNodes".cm.axisCommand.cathodeMainPnP1AxisY.posAbsolute[4] AND NOT "Unit1.Em5.ControlNodes".cm.axisCommand.cathodeMainPnP1AxisY.posAbsolute[5]);
END_REGION

REGION Network 105: CmCathodeMainPnP1AxisY Position Absolute Position
   RUNG wire#powerrail
      Contact( "Unit1.Em5.ControlNodes".cm.axisCommand.cathodeMainPnP1AxisY.posAbsoluteSummary )
      Coil( "Unit1.Em5.ControlNodes".cmCathodeMainPnP1AxisY.commands.posAbsolute )
   END_RUNG
   // the same network as SCL:
   "Unit1.Em5.ControlNodes".cmCathodeMainPnP1AxisY.commands.posAbsolute := "Unit1.Em5.ControlNodes".cm.axisCommand.cathodeMainPnP1AxisY.posAbsoluteSummary;
END_REGION

REGION Network 106: CmCathodeMainPnP2AxisY Interlock Summary
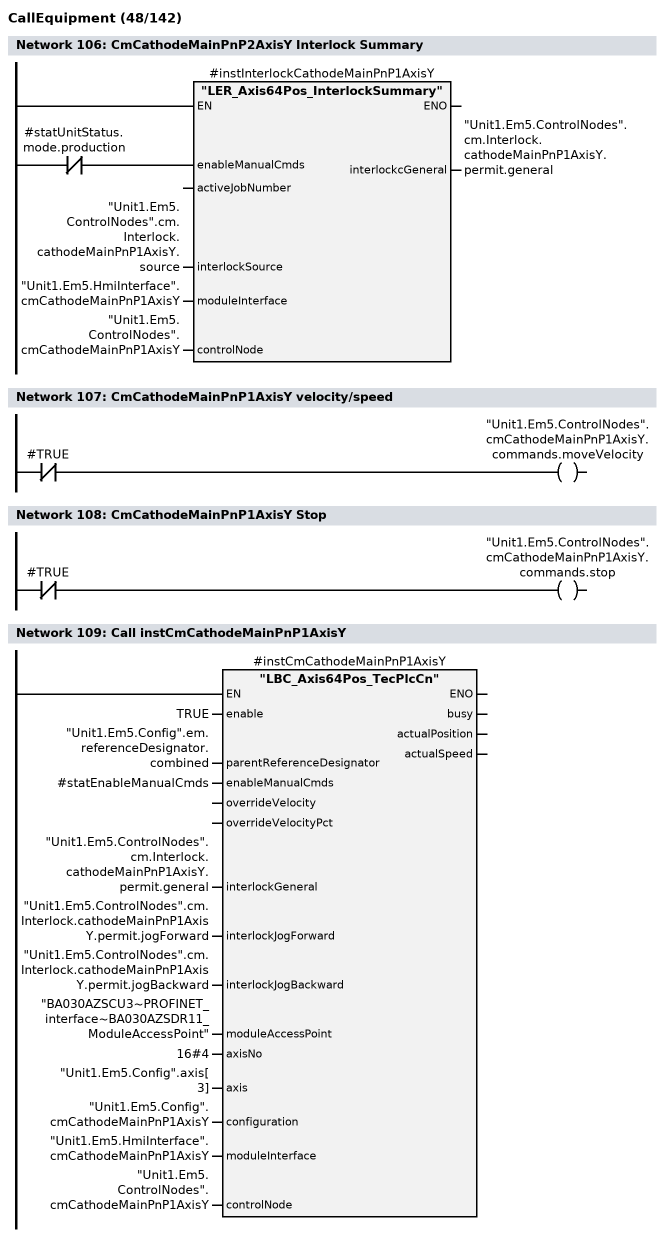
   RUNG wire#powerrail
      #instInterlockCathodeMainPnP1AxisY(enableManualCmds := wire#w1, activeJobNumber :=, interlockSource := "Unit1.Em5.ControlNodes".cm.Interlock.cathodeMainPnP1AxisY.source, moduleInterface := "Unit1.Em5.HmiInterface".cmCathodeMainPnP1AxisY, controlNode := "Unit1.Em5.ControlNodes".cmCathodeMainPnP1AxisY, interlockcGeneral => "Unit1.Em5.ControlNodes".cm.Interlock.cathodeMainPnP1AxisY.permit.general)
   END_RUNG
   RUNG wire#powerrail
      I_Contact( #statUnitStatus.mode.production )
   END_RUNG wire#w1
   // the same network as SCL:
   #instInterlockCathodeMainPnP1AxisY(enableManualCmds := NOT #statUnitStatus.mode.production,   // "LER_Axis64Pos_InterlockSummary"
                           interlockSource := "Unit1.Em5.ControlNodes".cm.Interlock.cathodeMainPnP1AxisY.source,
                           moduleInterface := "Unit1.Em5.HmiInterface".cmCathodeMainPnP1AxisY,
                           controlNode := "Unit1.Em5.ControlNodes".cmCathodeMainPnP1AxisY,
                           interlockcGeneral => "Unit1.Em5.ControlNodes".cm.Interlock.cathodeMainPnP1AxisY.permit.general);
END_REGION

REGION Network 107: CmCathodeMainPnP1AxisY velocity/speed
   RUNG wire#powerrail
      I_Contact( #TRUE )
      Coil( "Unit1.Em5.ControlNodes".cmCathodeMainPnP1AxisY.commands.moveVelocity )
   END_RUNG
   // the same network as SCL:
   "Unit1.Em5.ControlNodes".cmCathodeMainPnP1AxisY.commands.moveVelocity := NOT #TRUE;
END_REGION

REGION Network 108: CmCathodeMainPnP1AxisY Stop
   RUNG wire#powerrail
      I_Contact( #TRUE )
      Coil( "Unit1.Em5.ControlNodes".cmCathodeMainPnP1AxisY.commands.stop )
   END_RUNG
   // the same network as SCL:
   "Unit1.Em5.ControlNodes".cmCathodeMainPnP1AxisY.commands.stop := NOT #TRUE;
END_REGION

REGION Network 109: Call instCmCathodeMainPnP1AxisY
   RUNG wire#powerrail
      #instCmCathodeMainPnP1AxisY(enable := TRUE, parentReferenceDesignator := "Unit1.Em5.Config".em.referenceDesignator.combined, enableManualCmds := #statEnableManualCmds, overrideVelocity :=, overrideVelocityPct :=, interlockGeneral := "Unit1.Em5.ControlNodes".cm.Interlock.cathodeMainPnP1AxisY.permit.general, interlockJogForward := "Unit1.Em5.ControlNodes".cm.Interlock.cathodeMainPnP1AxisY.permit.jogForward, interlockJogBackward := "Unit1.Em5.ControlNodes".cm.Interlock.cathodeMainPnP1AxisY.permit.jogBackward, moduleAccessPoint := "BA030AZSCU3~PROFINET_interface~BA030AZSDR11_ModuleAccessPoint", axisNo := 16#4, axis := "Unit1.Em5.Config".axis[3], configuration := "Unit1.Em5.Config".cmCathodeMainPnP1AxisY, moduleInterface := "Unit1.Em5.HmiInterface".cmCathodeMainPnP1AxisY, controlNode := "Unit1.Em5.ControlNodes".cmCathodeMainPnP1AxisY, busy =>, actualPosition =>, actualSpeed =>)
   END_RUNG
   // the same network as SCL:
   #instCmCathodeMainPnP1AxisY(enable := TRUE,   // "LBC_Axis64Pos_TecPlcCn"
                           parentReferenceDesignator := "Unit1.Em5.Config".em.referenceDesignator.combined,
                           enableManualCmds := #statEnableManualCmds,
                           interlockGeneral := "Unit1.Em5.ControlNodes".cm.Interlock.cathodeMainPnP1AxisY.permit.general,
                           interlockJogForward := "Unit1.Em5.ControlNodes".cm.Interlock.cathodeMainPnP1AxisY.permit.jogForward,
                           interlockJogBackward := "Unit1.Em5.ControlNodes".cm.Interlock.cathodeMainPnP1AxisY.permit.jogBackward,
                           moduleAccessPoint := "BA030AZSCU3~PROFINET_interface~BA030AZSDR11_ModuleAccessPoint",
                           axisNo := 16#4,
                           axis := "Unit1.Em5.Config".axis[3],
                           configuration := "Unit1.Em5.Config".cmCathodeMainPnP1AxisY,
                           moduleInterface := "Unit1.Em5.HmiInterface".cmCathodeMainPnP1AxisY,
                           controlNode := "Unit1.Em5.ControlNodes".cmCathodeMainPnP1AxisY);
END_REGION

REGION Network 110: CmCathodeMainPnP1AxisY SoftCam
